# B&R Automation Studio project perfxxl (part 7)

#### referenz.c
```c
#ifdef _DEFAULT_INCLUDES
	#include <AsDefault.h>
#endif
/****************************************************************************/
/*	Ablauf Referenzfahrt */
/*																			*/
/*																			*/
/*	Versionsgeschichte:														*/
/*  Version		Datum		Änderung								von		*/
/*	1.00		25.09.02	erste Implementation					HA		*/
/*	*/
/*		*/
/*																			*/
/****************************************************************************/

#include "glob_var.h"
#include "in_out.h"
#include "standard.h"
#include "motorfunc.h"
#include "auxfunc.h"

#define ROT 0x002D
#define GRUEN 0x000A
#define GRAU 0x0007
#define GRAU59 0x003B
#define SCHWARZ 0x0000
#define WEISS 0x1010

#define RAHMEN_ROT 0x2D00
#define RAHMEN_SCHWARZ 0x0000
#define RAHMEN_GRAU 0x0700

_LOCAL	USINT	ReferenceStep;
_LOCAL TON_10ms_typ ReferenceTimer,CoverLockTimer;
TP_10ms_typ ColorTimer;

_LOCAL	UINT	FeederVerticalColor;
_LOCAL	UINT	FeederHorizontalColor;
_LOCAL	UINT	PaperRemoveVerticalColor;
_LOCAL	UINT	PaperRemoveHorizontalColor;
_LOCAL	UINT	DeloaderHorizontalColor;
_LOCAL	UINT	DeloaderTurnColor;
_LOCAL	UINT	FUColor;
BOOL	ColorToggle;
BOOL	DeloaderReady;
_GLOBAL	UINT	ConveyorBeltOn;
UDINT OriginalDeloaderRefSpeed;
_GLOBAL USINT	ClearLine;
_GLOBAL BOOL	DontCloseTrolley;
/*V1.95 sequenzen disablen, solange Fehlplatte abgeworfen wird*/
_GLOBAL BOOL	DisablePaperRemove;
_GLOBAL UINT MainPicNumber;

static    USINT               PinsStep;       /* holds current step of fct AdjPins */
static    TON_10ms_typ        PinsTimer;

_INIT void Init(void)
{
	PinsStep = 0;
	PinsTimer.IN = FALSE;
	ColorToggle = 0;
	ColorTimer.IN = 1;
	ReferenceStep = 0;
	ReferenceStart = 0;
	ReferenceTimer.IN = 0;
	ReferenceTimer.PT = 1;
	CoverLockTimer.IN = 0;
}

_CYCLIC void Cyclic(void)
{

	SequenceSteps[8] = ReferenceStep;

	TON_10ms(&PinsTimer);

	TON_10ms(&ReferenceTimer);
	TON_10ms(&CoverLockTimer);

	if (!ReferenceStart) ReferenceStep = 0;

	switch (ReferenceStep)
	{
		case 0:
		{

/* wait for start command */
			if (!ReferenceStart) break;

			if(	Motors[FEEDER_VERTICAL].Error
			||	(Motors[FEEDER_HORIZONTAL].Error && GlobalParameter.FlexibleFeeder)
			||	Motors[PAPERREMOVE_VERTICAL].Error
			||	Motors[PAPERREMOVE_VERTICAL2].Error
			||	Motors[PAPERREMOVE_HORIZONTAL].Error
			||	(Motors[DELOADER_HORIZONTAL].Error && GlobalParameter.DeloaderTurnStation>0)
			||	(Motors[DELOADER_TURN].Error && GlobalParameter.DeloaderTurnStation==2) )
			{
				ReferenceStart = 0;
				break;
			}
			ReferenceStep = 100;
			break;
		}

		case 2:
		{

			START = 0;
			PlateTakingStart = 0;
			PaperRemoveStart = 0;
			AdjustStart = 0;
			DeloadStart = 0;
			ExposeStart = 0;
			OpenTrolleyStart = 0;
			CloseTrolleyStart = 0;

			ClearStation(&PlateAtFeeder);
			AdjustReady = 0;
			ExposureReady = 0;
			DeloadReady = 0;
			ClearLine = 0;
			PlateTransportSim = 0;

			Motors[FEEDER_VERTICAL].ReferenceOk = 0;
			Motors[FEEDER_HORIZONTAL].ReferenceOk = 0;
			Motors[PAPERREMOVE_VERTICAL].ReferenceOk = 0;
			Motors[PAPERREMOVE_VERTICAL2].ReferenceOk = 0;
			Motors[PAPERREMOVE_HORIZONTAL].ReferenceOk = 0;
			Motors[DELOADER_HORIZONTAL].ReferenceOk = 0;
			Motors[DELOADER_TURN].ReferenceOk = 0;
			DeloaderReady = 0;
			ReferenceStep = 5;

			break;
		}
		case 5:
		{
			int i;
/*Feeder vacuum off and Feeder vert. reference*/
			for(i=0;i<5;i++)
				Out_FeederVacuumOn[i] = OFF;

			SwitchAdjustTableVacuum(0,ALL,OFF);
			AdjustBlowairOn = 0;
			Out_AdjustSuckerVacuumOn[0] = OFF;
			Out_AdjustSuckerVacuumOn[1] = OFF;
			Out_AdjustSuckerVacuumOn[2] = OFF;
			Out_AdjustSignalCross = OFF;
			Out_LiftingPinsUp = OFF;
			Out_LiftingPinsDown = ON;

			Motors[FEEDER_VERTICAL].StartRef = 1;

/*Deloader Horiz. pre reference very slowly*/
			if(GlobalParameter.DeloaderTurnStation>0)
			{
				Motors[DELOADER_HORIZONTAL].StartRef = 1;
/*HA 02.08.04 V1.80 bugfix: if no turning motor, do not set slow speed*/
				if (GlobalParameter.DeloaderTurnStation==2)
				{
					OriginalDeloaderRefSpeed = Motors[DELOADER_HORIZONTAL].Parameter.ReferenceSpeed;
					Motors[DELOADER_HORIZONTAL].Parameter.ReferenceSpeed = Motors[DELOADER_HORIZONTAL].Parameter.ReferenceSpeed / 2;
				}
			}
			ReferenceStep = 7;
			break;
		}

		case 7:
		{
			if(AdjPins(PINS_DOWN,&PinsStep,&PinsTimer))
				ReferenceStep = 10;
			break;
		}

		case 10:
		{
/*wait for Feeder vert. ref ready, then Feeder Horiz. ref*/

/*if deloader hor is ready, start turn*/
			if(GlobalParameter.DeloaderTurnStation==2)
			{
				if(Motors[DELOADER_HORIZONTAL].ReferenceOk && !Motors[DELOADER_TURN].ReferenceOk)
				{
					Motors[DELOADER_TURN].StartRef = 1;
				}
			}

			if( Motors[FEEDER_VERTICAL].ReferenceOk )
			{
				Out_FeederHorActive = OFF;
				Out_AdjustSuckerActive[0] = OFF;
				Out_AdjustSuckerActive[1] = OFF;
				Out_AdjustSuckerActive[2] = OFF;
				if(GlobalParameter.FlexibleFeeder)
					Motors[FEEDER_HORIZONTAL].StartRef = 1;

				Motors[PAPERREMOVE_VERTICAL].StartRef = 1;
				ReferenceStep = 11;
				break;
			}
			break;
		}

		case 11:
		{
/*X ok? -> start reference*/
			if( !FU.Error && !FU.CANError && FU.ENPO)
			{
				FU.cmd_Ref = 1;
/*wait for reference to start*/
				if(!FU.RefOk)
					ReferenceStep = 12;
			}
			else
				ReferenceStep = 12;
			break;
		}

		case 12:
		{
/*both motors ref ok? -> go on*/
			if(Motors[PAPERREMOVE_VERTICAL].ReferenceOk && Motors[PAPERREMOVE_VERTICAL2].ReferenceOk)
			{
				ReferenceStep = 15;
				break;
			}
/*wait for 1st motor, then start 2nd to avoid current peak*/
			if(Motors[PAPERREMOVE_VERTICAL].ReferenceOk)
			{
				Motors[PAPERREMOVE_VERTICAL2].StartRef = 1;
			}
			break;
		}

		case 15:
		{
/*wait for Feeder Horiz ref  ready, then paper remove vert ref */
/*if deloader hor is ready, start turn*/
			if(GlobalParameter.DeloaderTurnStation==2)
			{
				if(Motors[DELOADER_HORIZONTAL].ReferenceOk && !Motors[DELOADER_TURN].ReferenceOk)
				{
					Motors[DELOADER_TURN].StartRef = 1;
				}
			}
/*if Paperremove vertical ready start horiz*/
			if( Motors[PAPERREMOVE_VERTICAL].ReferenceOk && Motors[PAPERREMOVE_VERTICAL2].ReferenceOk && !Motors[PAPERREMOVE_HORIZONTAL].ReferenceOk )
			{
				Motors[PAPERREMOVE_HORIZONTAL].StartRef = 1;
			}

			if( (Motors[FEEDER_HORIZONTAL].ReferenceOk || !GlobalParameter.FlexibleFeeder) )
			{

				ReferenceStep = 20;
				break;
			}
			break;
		}
		case 20:
		{
/*if deloader hor is ready, start turn*/
			if(GlobalParameter.DeloaderTurnStation==2)
			{
				if(Motors[DELOADER_HORIZONTAL].ReferenceOk && !Motors[DELOADER_TURN].ReferenceOk)
				{
					Motors[DELOADER_TURN].StartRef = 1;
				}
			}

/*wait for Paperrem vert ref ready, then paper remove horiz. ref */
			if( Motors[PAPERREMOVE_VERTICAL].ReferenceOk && Motors[PAPERREMOVE_VERTICAL2].ReferenceOk )
			{
				if( !Motors[PAPERREMOVE_HORIZONTAL].ReferenceOk )
					Motors[PAPERREMOVE_HORIZONTAL].StartRef = 1;
				ReferenceStep = 22;
				break;
			}
			break;
		}
		case 22:
		{

/*if deloader hor is ready, start turn*/
			if(GlobalParameter.DeloaderTurnStation==2)
			{
				if(Motors[DELOADER_HORIZONTAL].ReferenceOk && !Motors[DELOADER_TURN].ReferenceOk)
				{
					Motors[DELOADER_TURN].StartRef = 1;
				}
			}

/*if deloader turn is ready, start hor again*/
			if(GlobalParameter.DeloaderTurnStation==2)
			{
				if(Motors[DELOADER_TURN].ReferenceOk)
				{
					Motors[DELOADER_HORIZONTAL].Parameter.ReferenceSpeed = OriginalDeloaderRefSpeed;
					Motors[DELOADER_HORIZONTAL].ReferenceOk = 0;
					Motors[DELOADER_HORIZONTAL].StartRef = 1;
					ReferenceStep = 23;
				}
			}
			else
				ReferenceStep = 23;

			break;
		}

		case 23:
		{
/*wait for Paperremove horiz. ref ready*/
			if(Motors[PAPERREMOVE_HORIZONTAL].ReferenceOk)
			{
				Out_PaperGripOn[LEFT] = OFF;
				Out_PaperGripOn[RIGHT] = OFF;
				ReferenceStep = 25;
			}
			break;
		}

		case 25:
		{

			switch (GlobalParameter.DeloaderTurnStation)
			{
				case 0:
				{
					ReferenceStep = 45;
					break;
				}
				case 1:
				{
					if (Motors[DELOADER_HORIZONTAL].ReferenceOk)
						ReferenceStep = 45;
					break;
				}
				case 2:
				{
					if (Motors[DELOADER_HORIZONTAL].ReferenceOk && Motors[DELOADER_TURN].ReferenceOk)
						ReferenceStep = 45;
					break;
				}
			}
			break;
		}
		case 45:
		{
/*X ok? -> check if ref ready*/
			if( !FU.Error && !FU.CANError && FU.ENPO)
			{
				if(FU.RefOk)
				{
					ReferenceStep = 46;
				}
			}
/*X not ok? ->ready*/
			else
			{
				ReferenceStep = 50;
			}
			break;
		}

/*HA 10.04.03 new steps 46 and 47 to move to axis parkpos after reference ok*/
/*move X to parkposition*/
		case 46:
		{
			FU.cmd_Park = 1;
			ReferenceStep = 47;
			break;
		}

/*wait for parkposition ready*/
		case 47:
		{
			if(FU.cmd_Park) break;
			ReferenceStep = 50;
			break;
		}

		case 50:
		{
/* Stop Conveyor Belt, Adjuster down */
			if(SendMotorCmd(CONVEYORBELT,"V0",0,0))
			{
				ReferenceStep = 57;
				ConveyorBeltOn = 0;
			}
			break;
		}
		case 57:
		{
			if(!Motors[CONVEYORBELT].Error)
				Motors[CONVEYORBELT].StartRef = 1;

			if( TCPConnected )
				BeamOFF = TRUE;

			ReferenceStep = 60;
			break;
		}
		case 60:
		{
			ClearStation(&PlateAtFeeder);
			AdjustReady = 0;
			ExposureReady = 0;
			DeloadReady = 0;
			PaperRemoveReady = 0;
			ReferenceStep = 0;
			ReferenceStart = 0;
			DontCloseTrolley = 0;
			DisablePaperRemove = 0;
			if(wBildNr == 26)
				wBildNeu = 1;
			break;
		}
/****************************************************************************/
/* HA 26.06.03 V1.11*/
/* SPECIAL STEPS FOR COVER LOCKING/CHECK */
/****************************************************************************/
		case 100:
		{
			if( DoorsOK || UserLevel>=1)
			{
				ReferenceStep = 104;
				CoverLockTimer.IN = 0;
				ReferenceTimer.IN = 0;
				break;
			}
			else
			{
				if(wBildAktuell != 41 )
					OrgBild = wBildAktuell;
				wBildNeu = 41;
				AbfrageOK = 0;
				AbfrageCancel = 0;
				IgnoreButtons = 0;
				OK_CancelButtonInv = 1;
				OK_ButtonInv = 0;
				AbfrageText1 = 43;
				AbfrageText2 = 44;
				AbfrageText3 = 0;
				AbfrageIcon = CAUTION;
				ReferenceStep = 106;
			}
			break;
		}

		case 104:
		{
/*timeout*/
			if( ReferenceTimer.Q )
			{
				CoverLockTimer.IN = 0;
				ReferenceTimer.IN = 0;
				ReferenceStep = 105;
				Out_CoverLockOn = 0;
				break;
			}
/*OK signal in time, or servicelevel 2*/
			if( CoverLockTimer.Q || UserLevel>=1 )
			{
				CoverLockTimer.IN = 0;
				ReferenceTimer.IN = 0;
				ReferenceStep = 2;
				break;
			}
			Out_CoverLockOn = 1;
			CoverLockTimer.IN = CoverLockOK && DoorsOK;
			CoverLockTimer.PT = 100;
			ReferenceTimer.IN = 1;
			ReferenceTimer.PT = 200;
			break;
		}

		case 105:
		{
				if(wBildAktuell != 41 )
					OrgBild = wBildAktuell;
				wBildNeu = 41;
				AbfrageOK = 0;
				AbfrageCancel = 0;
				IgnoreButtons = 0;
				OK_CancelButtonInv = 1;
				OK_ButtonInv = 0;
				AbfrageText1 = 41;
				AbfrageText2 = 42;
				AbfrageText3 = 0;
				AbfrageIcon = CAUTION;
				ReferenceStep = 106;
			break;
		}
/*wait for input */
		case 106:
		{
			if(AbfrageOK)
			{
				AbfrageOK = 0;
				ReferenceStep = 0;
				ReferenceStart = 0;
			}
			break;
		}

	} /*switch*/

/*colors for "LEDs"*/
	ColorTimer.PT = 50;

	if( ColorTimer.IN == 1 && ColorTimer.Q==1)
		ColorTimer.IN = 0;

	if( ColorTimer.IN == 0 && ColorTimer.Q==0)
	{
		ColorToggle = !ColorToggle;
		ColorTimer.IN = 1;
	}

	TP_10ms(&ColorTimer);

	if( Motors[FEEDER_VERTICAL].ReferenceOk)
	{
		FeederVerticalColor = SCHWARZ;
	}
	else
	{
		if(Motors[FEEDER_VERTICAL].Error)
			FeederVerticalColor = GRAU59;
		else
			if(Motors[FEEDER_VERTICAL].StartRef)
			{
				if(ColorToggle)
					FeederVerticalColor = SCHWARZ;
				else
					FeederVerticalColor = WEISS;
			}
			else /*no ref and ref not running*/
				FeederVerticalColor = WEISS;
	}

/*HA 20.01.04 V1.73 */
	if (!GlobalParameter.FlexibleFeeder)
		FeederHorizontalColor = WEISS;
	else
/*END HA 20.01.04 V1.73 */
	if( Motors[FEEDER_HORIZONTAL].ReferenceOk)
	{
		FeederHorizontalColor = SCHWARZ;
	}
	else
	{
		if(Motors[FEEDER_HORIZONTAL].Error)
			FeederHorizontalColor = GRAU59;
		else
			if(Motors[FEEDER_HORIZONTAL].StartRef)
			{
				if(ColorToggle)
					FeederHorizontalColor = SCHWARZ;
				else
					FeederHorizontalColor = WEISS;
			}
			else /*no ref and ref not running*/
				FeederHorizontalColor = WEISS;
	}

	if( Motors[PAPERREMOVE_HORIZONTAL].ReferenceOk)
	{
		PaperRemoveHorizontalColor = SCHWARZ;
	}
	else
	{
		if(Motors[PAPERREMOVE_HORIZONTAL].Error)
			PaperRemoveHorizontalColor = GRAU59;
		else
			if(Motors[PAPERREMOVE_HORIZONTAL].StartRef)
			{
				if(ColorToggle)
					PaperRemoveHorizontalColor = SCHWARZ;
				else
					PaperRemoveHorizontalColor = WEISS;
			}
			else /*no ref and ref not running*/
				PaperRemoveHorizontalColor = WEISS;
	}

	if( Motors[PAPERREMOVE_VERTICAL].ReferenceOk)
	{
		PaperRemoveVerticalColor = SCHWARZ;
	}
	else
	{
		if(Motors[PAPERREMOVE_VERTICAL].Error)
			PaperRemoveVerticalColor = GRAU59;
		else
			if(Motors[PAPERREMOVE_VERTICAL].StartRef)
			{
				if(ColorToggle)
					PaperRemoveVerticalColor = SCHWARZ;
				else
					PaperRemoveVerticalColor = WEISS;
			}
			else /*no ref and ref not running*/
				PaperRemoveVerticalColor = WEISS;
	}

/*HA 20.01.04 V1.73 */
	if (!GlobalParameter.DeloaderTurnStation)
		DeloaderHorizontalColor = WEISS;
	else
/*END HA 20.01.04 V1.73 */
	if( Motors[DELOADER_HORIZONTAL].ReferenceOk)
	{
		DeloaderHorizontalColor = SCHWARZ;
	}
	else
	{
		if(Motors[DELOADER_HORIZONTAL].Error && GlobalParameter.DeloaderTurnStation)
			DeloaderHorizontalColor = GRAU59;
		else
			if(Motors[DELOADER_HORIZONTAL].StartRef)
			{
				if(ColorToggle)
					DeloaderHorizontalColor = SCHWARZ;
				else
					DeloaderHorizontalColor = WEISS;
			}
			else /*no ref and ref not running*/
				DeloaderHorizontalColor = WEISS;
	}

/*HA 20.01.04 V1.73 */
	if (GlobalParameter.DeloaderTurnStation!=2)
		DeloaderTurnColor = WEISS;
	else
/*END HA 20.01.04 V1.73 */
	if( Motors[DELOADER_TURN].ReferenceOk)
	{
		DeloaderTurnColor = SCHWARZ;
	}
	else
	{
		if(Motors[DELOADER_TURN].Error)
			DeloaderTurnColor = GRAU59;
		else
			if(Motors[DELOADER_TURN].StartRef)
			{
				if(ColorToggle)
					DeloaderTurnColor = SCHWARZ;
				else
					DeloaderTurnColor = WEISS;
			}
			else /*no ref and ref not running*/
				DeloaderTurnColor = WEISS;
	}

	if(FU.Error || FU.CANError)
		FUColor = GRAU59;
	else
	if(FU.cmd_Ref && !FU.RefOk)
	{
		if (ColorToggle)
			FUColor = SCHWARZ;
		else
			FUColor = WEISS;
	}
	else
		if(FU.RefOk)
			FUColor = SCHWARZ;
		else
			FUColor = WEISS;

}
```

- motorfunc.h (reference to Logical/GlobalIncludes/motorfunc.h)

#### motorfunc.c
```c
#ifdef _DEFAULT_INCLUDES
	#include <AsDefault.h>
#endif
/*
                             *******************
******************************* C SOURCE FILE *******************************
**                           *******************                           **
**                                                                         **
** project  : LS JET II                                                    **
** filename : MOTORFUNC.C                                                  **
** version  : 1.02                                                         **
** date     : 07.11.2007                                                   **
**                                                                         **
*****************************************************************************
** Abstract                                                                **
** ========                                                                **
** Implementation of motor control functions (sending commands and         **
** check for positions)                                                    **
**                                                                         **
** Copyright (c) 2007, Krause-Biagosch GmbH                                **
** All rights reserved.                                                    **
**                                                                         **
*****************************************************************************
VERSION HISTORY:
----------------
Version     : 1.00
Date        : 20.10.2006
Revised by  : Herbert Aden
Description : Original version.

Version     : 1.01
Date        : 12.10.2007
Revised by  : Herbert Aden
Description : - a variable for holding the current step in function MoveToAbsPosition
                must now be provided by the caller (a pointer to that var of course!)
              - in Fct. IsPositionOK the check for being in a certain position window
                failed, if that window was 0, i.e. if an exact position is to be found
                the expression "currpos - checkpos < deviation" results in false, so it
                was changed to "currpos - checkpos <= deviation" so that if
                currpos==checkpos the result is still true for deviaition==0

Version     : 1.02
Date        : 07.11.2007
Revised by  : Herbert Aden
Description : - bugfix: in RequestMotorData the var SerialCmd.Request was set TRUE
                unconditionally. Caused sporadic Errormessages for serial comm.

*/
#define _MOTORFUNC_C_SRC

/****************************************************************************/
/**                                                                        **/
/**                           INCLUDE FILES                                **/
/**                                                                        **/
/****************************************************************************/
#include <stdlib.h>
#include <string.h>
#include "glob_var.h"
#include "motorfunc.h"

/****************************************************************************/
/**                                                                        **/
/**                       DEFINITIONS AND MACROS                           **/
/**                                                                        **/
/****************************************************************************/
/* NONE */

/****************************************************************************/
/**                                                                        **/
/**                      EXPORTED VARIABLES                                **/
/**                                                                        **/
/****************************************************************************/
/*@checked@*/
_GLOBAL   SerialCmd_Typ       SerialCmd;

/****************************************************************************/
/**                                                                        **/
/**                           GLOBAL VARIABLES                             **/
/**                                                                        **/
/****************************************************************************/
static  BOOL                  Send1Ready = 0;

/****************************************************************************/
/**                                                                        **/
/**                          EXPORTED FUNCTIONS                            **/
/**                                                                        **/
/****************************************************************************/

/****************************************************************************/
/** Send commands to a motor                                                */
/****************************************************************************/
BOOL	SendMotorCmd(const INT pMotor,const char *CmdStr,const BOOL UseValue,const DINT Value)
{
	if(SerialCmd.Send == FALSE) /*wait, till no other sending active*/
	{
		strcpy(SerialCmd.CmdString,CmdStr);
		SerialCmd.UseParameter = UseValue;
		SerialCmd.Parameter = Value;
		if (   (STREQ(CmdStr,CMD_ABSOLUTE_POS))
			|| (STREQ(CmdStr,CMD_RELATIVE_POS))
			|| (STREQ(CmdStr,CMD_MOVE_AT))
		  ) /*bei LA oder LR oder V Refdir verwenden, sonst nicht*/
			SerialCmd.UseRefDirection = TRUE;
		else
			SerialCmd.UseRefDirection = FALSE;

		SerialCmd.SendMotor = pMotor;
		SerialCmd.Send = TRUE;
		return TRUE;
	}
	else
		return FALSE;
}

/****************************************************************************/
/** Request data from a motor                                                */
/****************************************************************************/
BOOL	RequestMotorData(const INT pMotor,const char *CmdString)
{
	if( SerialCmd.Send == TRUE )
		return FALSE;
	else
	{
		SerialCmd.Request = TRUE;
		return SendMotorCmd(pMotor,CmdString,FALSE,0);
	}
}

/****************************************************************************/
/** Check, if a motor is in a certain position window                       */
/****************************************************************************/
BOOL	isPositionOk(const INT Motor,const DINT Pos,const DINT Deviation)
{
	DINT tmp;
	if (labs(Deviation) > 0 )
		tmp = labs(Deviation);
	else	/* if Dev is 0, then use deviation defined in motorparam*/
		tmp = labs(Motors[Motor].Parameter.PositionWindow);

	if( labs( labs(Motors[Motor].Position) - labs(Pos) ) <= tmp )
		return TRUE;
	else
		return FALSE;
}

/****************************************************************************/
/** Check, if a motor is below a certain position                           */
/****************************************************************************/
BOOL	isPositionLowerThan(const INT Motor,DINT Pos)
{
	if( labs(Motors[Motor].Position) < (labs(Pos) ) )
		return TRUE;
	else
		return FALSE;
}

/****************************************************************************/
/** Check, if a motor is above a certain position                           */
/****************************************************************************/
BOOL	isPositionHigherThan(const INT Motor,DINT Pos)
{
	if( labs(Motors[Motor].Position) > (labs(Pos) ) )
		return TRUE;
	else
		return FALSE;
}

/****************************************************************************/
/* send commands to paper remove vertical */
/****************************************************************************/
BOOL	PapRemVerticalCmd(BOOL Config,char *CmdString,BOOL UseValue,DINT Value)
{
	if(Config == LEFT)
		return SendMotorCmd(PAPERREMOVE_VERTICAL, CmdString, UseValue, Value);
	else
	if(Config == RIGHT)
		return SendMotorCmd(PAPERREMOVE_VERTICAL2, CmdString, UseValue, Value);
	else
	if ( Send1Ready == FALSE )
	{
		if( SendMotorCmd(PAPERREMOVE_VERTICAL, CmdString, UseValue, Value) )
			Send1Ready = TRUE;

		return FALSE;
	}
	else
	{
		if( SendMotorCmd(PAPERREMOVE_VERTICAL2, CmdString, UseValue, Value) )
		{
			Send1Ready = FALSE;
			return TRUE;
		}
		return FALSE;
	}
}

/****************************************************************************/
/* Check position of paper remove vertical */
/****************************************************************************/
BOOL	isPapRemVerticalOk(BOOL Config,DINT Pos,UDINT MaxDeviation)
{
	if(Config == LEFT)
		return isPositionOk(PAPERREMOVE_VERTICAL, Pos, MaxDeviation);
	else
	if(Config == RIGHT)
		return isPositionOk(PAPERREMOVE_VERTICAL2, Pos, MaxDeviation);
	else
	if ( isPositionOk(PAPERREMOVE_VERTICAL, Pos, MaxDeviation) )
	{
		if ( isPositionOk(PAPERREMOVE_VERTICAL2, Pos, MaxDeviation) )
			return TRUE;
		else
			return FALSE;
	}
	else
		return FALSE;
}

/****************************************************************************/
/* move motor to an absolute position and wait for motion to start */
/****************************************************************************/
BOOL  MoveToAbsPosition(INT pMotor, DINT Pos, DINT Speed, USINT *pStep)
{
	int step = *pStep;

	BOOL retval = FALSE;

	if (pMotor == 0 && Pos == 0L && Speed == 0L)
	{
		step = 0;
		*pStep = 0;
		return FALSE;
	}

	switch (step)
	{
		case 0:
		{
/* send target position */
			if( SendMotorCmd(pMotor,CMD_ABSOLUTE_POS,TRUE,Pos) )
			{
				if ( Speed == DONT_SEND_SPEED )
					step = 20;
				else
					step = 10;
			}
			retval = FALSE;
			break;
		}
/* set speed */
		case 10:
		{
			if( SendMotorCmd(pMotor,CMD_SPEED,TRUE,Speed) )
			{
				step = 20;
			}
			retval = FALSE;
			break;
		}
		case 20:
		{
/* start motion */
			if( SendMotorCmd(pMotor,CMD_START_MOTION,FALSE,0L) )
			{
				step = 30;
			}
			retval = FALSE;
			break;
		}
		case 30:
		{
/* Wait til motion begins or Motor is in position (might be already there!)*/
			if( Motors[pMotor].Moving
			    ||
			    isPositionOk(pMotor,Pos,0) )
			{
				step = 0;
				retval = TRUE;
			}
			break;
		}
	}
	*pStep = step;
	return retval;
}

/****************************************************************************/
/* move motor to an relative position without waiting for motion to start */
/****************************************************************************/
BOOL  MoveToRelPosition(INT pMotor, DINT Pos, DINT Speed, USINT *pStep)
{
	int step = *pStep;

	BOOL retval = FALSE;

	if (pMotor == 0 && Pos == 0L && Speed == 0L)
	{
		step = 0;
		*pStep = 0;
		return FALSE;
	}

	switch (step)
	{
		case 0:
		{
/* send target position */
			if( SendMotorCmd(pMotor,CMD_RELATIVE_POS,TRUE,Pos) )
			{
				if ( Speed == DONT_SEND_SPEED )
					step = 20;
				else
					step = 10;
			}
			retval = FALSE;
			break;
		}
/* set speed */
		case 10:
		{
			if( SendMotorCmd(pMotor,CMD_SPEED,TRUE,Speed) )
			{
				step = 20;
			}
			retval = FALSE;
			break;
		}
		case 20:
		{
/* start motion */
			if( SendMotorCmd(pMotor,CMD_START_MOTION,FALSE,0L) )
			{
				step = 30;
			}
			retval = FALSE;
			break;
		}
		case 30:
		{
			step = 0;
			retval = TRUE;
			break;
		}
	}
	*pStep = step;
	return retval;
}

/****************************************************************************/
/**                                                                        **/
/**                          LOCAL FUNCTIONS                               **/
/**                                                                        **/
/****************************************************************************/
/* NONE */

/****************************************************************************/
/**                                                                        **/
/**                                 EOF                                    **/
/**                                                                        **/
/****************************************************************************/
```

- auxfunc.h (reference to Logical/GlobalIncludes/auxfunc.h)

### Program Logical/Exposer/Ablauf/expose (ANSIC, version 1.12.0) - Belichtungsablauf

#### belichten.c
```c
#ifdef _DEFAULT_INCLUDES
	#include <AsDefault.h>
#endif
/****************************************************************************/
/*	Ablauf belichten */
/*																			*/
/*																			*/
/*	Versionsgeschichte:														*/
/*  Version		Datum		Änderung								von		*/
/*	1.0			19.09.02	erste Implementation					HA		*/
/*	1.10		13.11.02	erweiterte TB1-Komm. (Polygonspeed)		HA		*/
/*	1.11		02.04.03	Belichtung wird im AUTO Modus nicht 	HA		*/
/*							gestartet, wenn keine Verbindung zum TIFFBlaster */
/*							und keine TB Simulation*/
/*	1.12		07.04.03	Ausgabe: Warte auf Daten..." implementiert 	HA		*/
/*																			*/
/*																			*/
/****************************************************************************/

#include "glob_var.h"
#include "asstring.h"
#include "sys_lib.h"
#include "in_out.h"
#include <string.h>

#define	MAXFILELIST	32
#define TCPIPTIMEOUT 150

_LOCAL	USINT	ExposeStep;
_LOCAL TON_10ms_typ ExposeTimer;
USINT			tmp[20];

_GLOBAL	STRING	FileName[100];
_GLOBAL	USINT	FileListShift;
_GLOBAL	STRING	FileListName[MAXFILELIST][50];
_GLOBAL	STRING	FileListStatus[MAXFILELIST][5];
_GLOBAL	STRING	FileListTime[MAXFILELIST][20];
_GLOBAL	STRING	FileListResolution[MAXFILELIST][5];

_GLOBAL BOOL	AdjustFailed;
_GLOBAL BOOL	ExposingStarted;	/*HA 08.07.03 V1.14 Flag to inform plate taking that exposing has started*/

_GLOBAL	RTCtime_typ	RTCtime;

_GLOBAL UDINT	PlatesMade;		/* [0] = Plates made ever,[1] = plates made today*/
_GLOBAL	UDINT	PlatesMadeToday;
_GLOBAL	BOOL	savePlatesMade;

_GLOBAL USINT	ClearLine;

_LOCAL	USINT	Length,PermanentMode;

int	TimeoutCounter,i;
BOOL	StepChanged;
_LOCAL UINT	ExposureProgress;
_GLOBAL 	BOOL	SendYOffset,SendLP,SendOSCommand;
STRING tmpstr[100];
int waitcounter;

_LOCAL    UINT                CheckForDataStep;
_LOCAL    USINT               TestNumberOfPlates,TestPlateType;
static    USINT               OldSecond;
_LOCAL    BOOL                StopCheckingForData;

_INIT void init(void)
{
	StepChanged = 0;
	ExposeStep		= 0;
	ExposeStart	= 0;
	ExposureReady		= 0;
	ExposeTimer.IN	= 0;
	ExposeTimer.PT	= 10; /*just to have any value in there...*/

	Expose_Param.ScansPerMinute			= 96000;
	Expose_Param.Resolution				= 1270;

	PlatesMadeToday = 0;
	ExposingStarted = 0;
	PermanentMode = 0;
	CheckForDataStep = 0;
	StopCheckingForData = 0;
	OldSecond = 0;
	TestPlateType = 1;
}

_CYCLIC void cyclic(void)
{
UINT RequiredLaserPower;

	SequenceSteps[4] = ExposeStep;

	TON_10ms(&ExposeTimer);

/*	if(START)*/
/*HA 28.05.03 V1.13 added "|| ClearLine" */
	if( (AdjustReady) && AUTO
		&& (GlobalParameter.TBSimulation || TCPConnected || ClearLine))
		 ExposeStart=1;

/*safety*/
	if( !ExposeStart )
	{
		 PermanentMode = 0;
		 ExposeStep = 0;
		 ExposingStarted = 0;
/*		 strcpy(FileName,"----");*/
		 ExposureProgress = 0;
	}

	switch (ExposeStep)
	{
		case 0:
		{
			if(!ExposeStart) break;

			ExposeStep = 2;
			break;
		}

		case 2:
		{
			REAL AccWay = 3.0;
			if (DisableTable || AdjustStart) break; /*SAFETY*/

/* for LSJet 350: if speed is > than the usual 97000 then double acceleration/deceleration way*/
			if(Expose_Param.ScansPerMinute < 99000)
				AccWay = 3.0;
			else
				AccWay = 6.0;

			Expose_Param.PEGStartPosition = PlateParameter.XOffset+PlateParameter.Length;
			if ( Expose_Param.PEGStartPosition > X_Param.MaxPosition ) Expose_Param.PEGStartPosition = X_Param.MaxPosition;
			Expose_Param.PEGEndPosition = PlateParameter.XOffset;
			if ( Expose_Param.PEGEndPosition < X_Param.MinPosition ) Expose_Param.PEGEndPosition = X_Param.MinPosition;
			Expose_Param.StartPosition = PlateParameter.XOffset+PlateParameter.Length + AccWay;
			if ( Expose_Param.StartPosition > X_Param.MaxPosition ) Expose_Param.StartPosition = X_Param.MaxPosition;
			Expose_Param.EndPosition = PlateParameter.XOffset - AccWay;
			if ( Expose_Param.EndPosition < X_Param.MinPosition ) Expose_Param.EndPosition = X_Param.MinPosition;

			if ( FU.cmd_Target == 0 )
			{
				FU.TargetPosition_mm = Expose_Param.StartPosition;
				FU.cmd_Target = 1;
				ExposeStep = 3;
			}
			break;
		}
		case 3:
		{
/*und warten*/
			if ( abs(FU.aktuellePosition_mm - FU.TargetPosition_mm )< 2 )
			{
/*Tisch ist in Position -> OK, weiter*/
				ExposeStep = 5;
			}
			break;
		}

		case 5:
		{
/* Communication with TiffBlaster*/
			if(GlobalParameter.TBSimulation || ClearLine)
			{
				strcpy(FileName,"KrauseTestImage.TIF");
				ExposeStep = 20;
				StepChanged = 1;
				break;
			}
/*Warte auf Daten...*/
			if (DataReady)
			{
				ExposeStep = 15;
				StepChanged = 1;
				StopCheckingForData = 1;
			}

			break;
		}

/*V2.15 automatische Laserleistungseinstellung bei Aufl Wechsel*/
		case 15:
		{
			if( AdjustFailed  )
			{
				ExposeStep	= 0;
				ExposeStart	= 0;
				break;
			}

/*
if plate is longer than 600 mm then wait for adjusting to finish,
to make sure, the plate cannot be under the beam during power setting
*/
			if(!AdjustReady && AUTO && (PlateParameter.Length>600))
				break;

/*Range check for safety*/
			if(Expose_Param.Resolution < 300 || Expose_Param.Resolution > 4000)
			{
				Expose_Param.Resolution=1270;
				GlobalParameter.Resolution = 1270;
			}

/*check, which laserpower to use*/
			RequiredLaserPower = GlobalParameter.RealLaserPower;
/*gehe durch die Liste, bis sie entweder ganz abgearbeitet ist oder die passende Aufl gefunden wurde*/
			for (i=1; i<MAXLASERPOWERSETTINGS ; i++)
			{
				if ( Expose_Param.Resolution == LaserPowerSettings[i].Resolution )
				{
/*if-construct for safety*/
					if ((PlateParameter.Number>0)&& (PlateParameter.Number<MAXPLATETYPES))
						RequiredLaserPower = LaserPowerSettings[i].LaserPower[PlateParameter.Number];
					else
						RequiredLaserPower = LaserPowerSettings[i].LaserPower[1];
					break;
				}
			}

/*if the power is different from currently used power, then send new power*/
			if (RequiredLaserPower != GlobalParameter.RealLaserPower)
			{
				GlobalParameter.RealLaserPower = RequiredLaserPower;
				SendLP = 1;
			}

/*go ahead if Power setting is ready or not started*/
			if ( !SendLP )
			{
				ExposeStep = 16;
/* HA V1.36 08.05.06 send Open Shutter command to TB*/
				SendOSCommand = 1;
				StepChanged = 1;
			}
			break;
		}

/* HA V2.10  08.05.06 send Open Shutter command to TB*/
		case 16:
		{
			waitcounter = 0;
			if (SendOSCommand == 0)
				ExposeStep = 18;
			break;
		}

/* wait shortly*/
		case 18:
		{
			waitcounter++;
			if (waitcounter >= 120)/*120 cycles = 0,6 sec*/
			{
				ExposeStep = 20;
				waitcounter = 0;
				StepChanged = 1;
			}
			break;
		}

		case 20:
		{
			if(StepChanged)
			{
				if(strlen(FileName)<50)
					strcpy(&FileListName[MAXFILELIST-1][0],FileName);
				else
				{
					memcpy(&FileListName[MAXFILELIST-1][0],FileName,48);
					FileListName[MAXFILELIST-1][49]=0;
				}
				itoa(Expose_Param.Resolution,(UDINT)&FileListResolution[MAXFILELIST-1][0]);
				strcpy(&FileListStatus[MAXFILELIST-1][0],"ACT");
				itoa(RTCtime.hour,(UDINT)&tmp[0]);
				if(RTCtime.hour<=9)
					strcpy(&FileListTime[MAXFILELIST-1][0],"0");
				else
					strcpy(&FileListTime[MAXFILELIST-1][0],"");
				strcat(&FileListTime[MAXFILELIST-1][0],&tmp[0]);
				strcat(&FileListTime[MAXFILELIST-1][0],":");
				itoa(RTCtime.minute,(UDINT)&tmp[0]);
				if(RTCtime.minute<=9)
					strcat(&FileListTime[MAXFILELIST-1][0],"0");
				strcat(&FileListTime[MAXFILELIST-1][0],&tmp[0]);
				strcat(&FileListTime[MAXFILELIST-1][0],":");
				itoa(RTCtime.second,(UDINT)&tmp[0]);
				if(RTCtime.second<=9)
					strcat(&FileListTime[MAXFILELIST-1][0],"0");
				strcat(&FileListTime[MAXFILELIST-1][0],&tmp[0]);
				StepChanged = 0;
				FileListShift = 1;
			}

			if(Expose_Param.Resolution < 300 || Expose_Param.Resolution > 4000)
			{
				Expose_Param.Resolution=1270;
				GlobalParameter.Resolution = 1270;
			}

			if(Expose_Param.ScansPerMinute<1000 || Expose_Param.ScansPerMinute>150000)
				Expose_Param.ScansPerMinute = 76200;

/*calculate X-speed*/
			Expose_Param.ExposeSpeed = (25.4/60.0) * ((REAL)Expose_Param.ScansPerMinute/(REAL)Expose_Param.Resolution);

			if(Expose_Param.ExposeSpeed<1 || Expose_Param.ExposeSpeed>100)
				Expose_Param.ExposeSpeed = 25.4;

/*wait for adjusting to finish*/
			if( AdjustReady || !AUTO)
			{
				FU.cmd_Expose = 1;
/*HA 08.07.03 V1.14 Flag to inform plate taking that exposing has started*/
				ExposingStarted = 1;
				ExposeStep = 25;
				StepChanged = 1;
			}

/*HA 17.02.04 V1.74B Adjusting failed and MaxFailedPlates is 0: stop */
			if( AdjustFailed && (AdjusterParameter.MaxFailedPlates == 0) )
			{
				ExposeStep	= 0;
				ExposeStart	= 0;
				break;
			}

			if( AdjustFailed && AUTO )
			{
				strcpy(&FileListStatus[0][0],"ERR");
				itoa(RTCtime.hour,(UDINT)&tmp[0]);
				if(RTCtime.hour<=9)
					strcpy(&FileListTime[0][0],"0");
				else
					strcpy(&FileListTime[0][0],"");
				strcat(&FileListTime[0][0],&tmp[0]);
				strcat(&FileListTime[0][0],":");
				itoa(RTCtime.minute,(UDINT)&tmp[0]);
				if(RTCtime.minute<=9)
					strcat(&FileListTime[0][0],"0");
				strcat(&FileListTime[0][0],&tmp[0]);
				strcat(&FileListTime[0][0],":");
				itoa(RTCtime.second,(UDINT)&tmp[0]);
				if(RTCtime.second<=9)
					strcat(&FileListTime[0][0],"0");
				strcat(&FileListTime[0][0],&tmp[0]);

				ExposureReady = 1;
				ExposeStep = 26;
			}
			break;
		}

		case 25:
		{
#ifdef PERFORMANCE
			if ((FU.aktuellePosition_mm <= Expose_Param.PEGStartPosition) && (PlateParameter.Length > 1))
			{
				ExposureProgress = ((Expose_Param.PEGStartPosition - FU.aktuellePosition_mm) *100.0)
									 / PlateParameter.Length;
			}
#else
			if ((FU.aktuellePosition_mm > Expose_Param.PEGStartPosition) && (PlateParameter.Length > 1))
			{
				ExposureProgress = ((FU.aktuellePosition_mm-Expose_Param.PEGStartPosition) *100.0)
									 / PlateParameter.Length;
			}
#endif
			else
				ExposureProgress = 0;
/*Wait for Exposure ready*/
			if(FU.cmd_Expose) break;
			if(!ExposureReady)
			{
				strcpy(&FileListStatus[0][0],"RDY");
				itoa(RTCtime.hour,(UDINT)&tmp[0]);
				if(RTCtime.hour<=9)
					strcpy(&FileListTime[0][0],"0");
				else
					strcpy(&FileListTime[0][0],"");
				strcat(&FileListTime[0][0],&tmp[0]);
				strcat(&FileListTime[0][0],":");
				itoa(RTCtime.minute,(UDINT)&tmp[0]);
				if(RTCtime.minute<=9)
					strcat(&FileListTime[0][0],"0");
				strcat(&FileListTime[0][0],&tmp[0]);
				strcat(&FileListTime[0][0],":");
				itoa(RTCtime.second,(UDINT)&tmp[0]);
				if(RTCtime.second<=9)
					strcat(&FileListTime[0][0],"0");
				strcat(&FileListTime[0][0],&tmp[0]);
				StepChanged = 0;
				PlatesMade++;
				PlatesMadeToday++;
				savePlatesMade=1;
			}
			ExposureReady = 1;
			ExposeStep = 26;
			ExposureProgress = 0;

			StopCheckingForData = 0;
			DataReady = 0;
			break;
		}
		case 26:
		{

/*feeder fährt runter: Tisch darf nicht fahren*/
			if (DisableTable)
				break;

/****************************************************************************/

/*wait for deloading ready, then go on*/
			if(DeloadReady || !AUTO)
			{
				DeloadReady = 0;
				ExposureReady = 0;
				ExposeStep = 30;
			}

			break;
		}
		case 30:
		{
			if ( PermanentMode && !AUTO )
				ExposeStep = 5;
			else
				ExposeStep = 35;
			break;
		}
		case 35:
		{
			ExposeStep = 0;
			ExposeStart = 0;
			break;
		}
	} /*switch*/

/****************************************************************************/
/* V2.50 asynchronous checking for data*/
/****************************************************************************/
	if( (ReferenceStart && (ExposeStep == 0))
	 || (ClearLine == TRUE)
	)
	{
		DataReady = 0;
		StopCheckingForData = 0;
		CheckForDataStep = 0;
	}

	if(GlobalParameter.TBSimulation)
	{
/* V2.55 Durchlaufsimulation*/
		DataReady = 1;
		TestNumberOfPlates = 3;

		if (TestNumberOfPlates==0)
			TestNumberOfPlates = 1;
		if (DataReady)
		{
			PlateToDo.PlateType = TestPlateType;
		}

	}

	switch (CheckForDataStep)
	{
		case 0:
		{
/*	check for data every second */
			if( (RTCtime.second != OldSecond)
			&& !StopCheckingForData
			&& !(GlobalParameter.TBSimulation || !TCPConnected)
			&& !ClearLine
			&& !SendLP
			&& !SendOSCommand
			&& !SendYOffset
			&& !ReferenceStart
			  )
				CheckForDataStep = 5;
			break;
		}
		case 5:
		{
/* Communication with TiffBlaster*/
			OldSecond = RTCtime.second;
			if(TCPSendCmd == 0)
			{
				strcpy(TCPCmd,"15");
				TCPSendCmd = 1;
				CheckForDataStep = 6;
			}
			TimeoutCounter = 0;
			break;
		}
		case 6:
		{

			if( !TCPRcvFlag)
			{
				TimeoutCounter++;
				if(TimeoutCounter>TCPIPTIMEOUT)
				{
					TimeoutCounter = 0;
					if(GlobalParameter.TBSimulation || !TCPConnected)
					{
						CheckForDataStep = 0;
						break;
					}

					CheckForDataStep = 0;
					DataReady = 0;
					switch (GlobalParameter.Language)
					{
						case 0:
						{
							strcpy(FileName,"Warte auf TIFF Blaster...");
							break;
						}
						case 1:
						{
							strcpy(FileName,"Waiting for TIFF Blaster...");
							break;
						}
					}
				}
				break;
			}

/*****       TCP answer received   *************/
/*IP0 : wait*/
			TCPRcvFlag = 0;
			if( TCPAnswer[2]=='0')
			{
				CheckForDataStep = 7;
				TimeoutCounter = 0;
				DataReady = 0;
				switch (GlobalParameter.Language)
				{
					case 1: /*deutsch*/
					{
						strcpy(FileName,"Warte auf Daten...");
						break;
					}
					default: /*english*/
					{
						strcpy(FileName,"Waiting for data...");
					}
				}
				break;
			}
			if(TCPAnswer[2]=='1')
			{
/* Aufbau des Strings:

Byte 0..2 	Fix: IP1
Byte 3..6 	Auflösung, fix 4stellig
Byte 7..12	Scans Pro Minute, fix 6stellig
Byte 13		Plattentyp
Byte 14		Anzahl Platten
Byte 15..End	Dateiname
BSP:	IP1127009600032C:\FileName.TIF
*/

				Length = strlen(TCPAnswer)-15;
				if(Length < 50 && Length>0 )
				{
			/*extract resolution*/
					memcpy(	tmp,&TCPAnswer[3],4 );
					tmp[4] = 0;
					Expose_Param.Resolution = atoi((UDINT) &tmp);
			/*extract Scans per min */
					memcpy(	tmp,&TCPAnswer[7],6 );
					tmp[6] = 0;
					Expose_Param.ScansPerMinute = atoi((UDINT) &tmp);
			/*extract Platetype */
					memcpy(	tmp,&TCPAnswer[13],1 );
					tmp[1] = 0;
			/*extract Number of plates */
					memcpy(	tmp,&TCPAnswer[14],1 );
					tmp[1] = 0;
			/*extract Filename */
					memcpy(	FileName,&TCPAnswer[15],Length );
					FileName[Length]=0;
				}
				CheckForDataStep = 0;
				DataReady = 1;
				StopCheckingForData = 1;
			}
			break;
		}

/*Warteschritt, um 14 etwas langsamer zu schicken*/
		case 7:
		{
/*Timeoutcounter hier als wartecounter missbraucht*/
			TimeoutCounter++;
			if(TimeoutCounter>20) /* 200 ms*/
			{
				TimeoutCounter = 0;
				CheckForDataStep = 5;
			}
			break;
		}
	}

}
```

### Program Logical/Exposer/Ablauf/entladen (ANSIC, version 1.30.0) - Platte Entladen aufs Transportband

#### entladen.c
```c
#ifdef _DEFAULT_INCLUDES
	#include <AsDefault.h>
#endif
/****************************************************************************/
/*	Ablauf Platte Entladen */
/*																						*/
/*																						*/
/*	Versionsgeschichte:																*/
/*  Version		Datum		Änderung										von		*/
/*	1.0			17.09.02	erste Implementation								HA		*/
/*																						*/
/*																						*/
/****************************************************************************/
#include "glob_var.h"
#include "asstring.h"
#include <string.h>
#include "in_out.h"
#include "Motorfunc.h"
#include "auxfunc.h"

#define CONVEYORBELT_BACKWAY	5000

_LOCAL	USINT	DeloadStep;
_LOCAL TON_10ms_typ DeloadTimer;
USINT			tmp[20];

_LOCAL TON_10ms_typ CycleTimer,CycleTimer2,TestTimer;
_LOCAL R_TRIGtyp R_TRIG_01;
_LOCAL F_TRIGtyp F_TRIG_01,F_TRIG_02;

BOOL	Started;
_GLOBAL UDINT PlatesPerHour;
/*HA 21.01.04 V1.73*/
_GLOBAL BOOL	AdjustFailed;

_LOCAL	UINT	CurrentTime;
_LOCAL	REAL	LastTime,HandlingTime;
DINT	Result1,Result2;
UDINT	TurnSpeedOld;
		TOF_10ms_typ	ConveyorBeltDelay;
		TON_10ms_typ	EGMErrorDelay;
		TON_10ms_typ	PinsDownWait;
		TON_10ms_typ	TurnOK;
		TOF_10ms_typ	ConveyorBeltSensorDelay1,ConveyorBeltSensorDelay2;

_GLOBAL	UINT			ConveyorBeltOn;

/*HA 14.01.04 V1.71 implemented Stop pins on conveyor */
_GLOBAL	BOOL			StopPinsUp;
		TON_10ms_typ	PinsDownDelay;
		TOF_10ms_typ	PinsUpDelay;

/*HA 05.09.03 V1.51 to avoid adjustsensor triggered by deloaded plate*/
/*HA 08.09.03 V1.52 disable-flags for right adjuster*/
_GLOBAL 	BOOL			DisableAdjustSensor,DisableAdjusterUp,EnableShuttle;
_LOCAL	BOOL			StartConveyorBelt,StopConveyorBelt;
		BOOL			LayOffPos2;
		UDINT			TempPlateReleasePosition,TempTurnPosition,TempTakePosition;

		REAL			PlateDeloadLength; /*holds calculated value Length*LengthFactor*/
BOOL TurnPosOK; /*Hilfsvariable für drehen ohne Zeit*/
_GLOBAL	BOOL	ConveyorbeltSimulation;
int DeloadSpeed,StopPinsStep;
BOOL	DisableConveyorBelt;
DINT ConveyorBeltPos,ConveyorBeltBack;
BOOL dummyflag;
USINT	ReturnStep;
_GLOBAL UINT	HideKrause;
USINT ConveyorBeltStep;
TON_10ms_typ	ConveyorBeltTimer;
UDINT	ConveyorTime;

_GLOBAL	REAL	TablePosDrop;
BOOL	MovingToParkpos,NoSpeedChange;
static USINT ConvMotStep;
TON_10ms_typ LiftpinsDownTimer;
static BOOL FirstTime;
static REAL OldParkSpeed;
static BOOL ParkSpeedChanged;

_LOCAL BOOL  JetValuesValid;
_LOCAL REAL  JetSqmValue; /* in m² for the plate set, i.e. no matter if 1 or 2 plates,
                             sum up must be done by jet */
_LOCAL USINT JetPlateCnt; /* 1 or 2 plates*/
static TON_10ms_typ JetValuesValidDelay;

void InformBluefin(void)
{
	if(!JetValuesValid)
	{
		if(PlateOnConveyorBelt.PlateConfig == BOTH)
			JetPlateCnt = 2;
		else
			JetPlateCnt = 1;

		if( (PlateOnConveyorBelt.PlateType > 0)
		 && (PlateOnConveyorBelt.PlateType < MAXPLATETYPES)
		  )
		{
/* /1000 weil Length und Width in mm sind, die Fläche aber in QadratMETER*/
			JetSqmValue = (PlateTypes[PlateOnConveyorBelt.PlateType].Length / 1000.0) *
			              (PlateTypes[PlateOnConveyorBelt.PlateType].Width / 1000.0);
				JetSqmValue *= JetPlateCnt;
		}
/* little delay to make sure the values are transmitted before the valid flag is set*/
		JetValuesValidDelay.IN = TRUE;
	}
	/* no else: Bluefin did not reset Valid-flag...do nothing */
}

_INIT void init(void)
{
	JetValuesValidDelay.IN = FALSE;
	JetValuesValid = FALSE;
	JetSqmValue = 0.0;
	JetPlateCnt = 1;
	ParkSpeedChanged = FALSE;
	FirstTime = TRUE;
	ConvMotStep = 0;
	LayOffPos2 = 0;
	ClearStation(&PlateOnConveyorBelt);
	DisableConveyorBelt = 0;
	StopPinsStep = 0;
	ClearStation(&PlateAtDeloader);
	TurnSpeedOld	= 0;
	DeloadStep		= 0;
	DeloadStart	= 0;
	DeloadReady		= 0;
	DeloadTimer.IN	= 0;
	DeloadTimer.PT	= 10; /*just to have any value in there...*/
	CycleTimer.IN	= 0;
	CycleTimer.PT	= 10; /*just to have any value in there...*/
	ConveyorBeltDelay.IN = 0;
	ConveyorBeltDelay.PT = 1000;
	ConveyorBeltOn = FALSE;
	EnableShuttle = 0;
	TurnOK.PT = 50;
	TurnOK.IN = 0;
	TurnPosOK = 0;
	LiftpinsDownTimer.IN = FALSE;

}

/****************************************************************************/
/* zyklischer Teil*/
/****************************************************************************/
_CYCLIC void cyclic(void)
{
#ifdef PERFORMANCE
	GlobalParameter.DeloaderTurnStation = 0;
#endif

	if( GlobalParameter.DisableSlowMode )
		SlowMode = 0;
	if( GlobalParameter.SlowModeWaitTime > 9900 )
		GlobalParameter.SlowModeWaitTime = 2000;

	SequenceSteps[5] = DeloadStep;

	if(ExposureReady && AUTO)
		DeloadStart = 1;

	TON_10ms(&DeloadTimer);
	TON_10ms(&TurnOK);

	LiftpinsDownTimer.IN = Out_LiftingPinsDown;
	LiftpinsDownTimer.PT = 12000; /* 2 min */
	TON_10ms(&LiftpinsDownTimer);

/* little delay for Bluefin comm handshake flag*/
	JetValuesValidDelay.PT = 15; /* 150ms */
	TON_10ms(&JetValuesValidDelay);
	if(JetValuesValidDelay.Q)
	{
		JetValuesValidDelay.IN = FALSE;
		JetValuesValid = TRUE;
	}
/* time measurement*/

/*detect edge of expose command*/
R_TRIG_01.CLK = FU.cmd_Expose;
R_TRIG(&R_TRIG_01);
if(R_TRIG_01.Q && Started)
{
	Started = 0;
	CycleTimer.IN = 0;
	Result1 = CycleTimer.ET;
	CycleTimer2.IN = 1;
	LastTime = (REAL)(Result1)/100.0;
	PlatesPerHour = (UDINT) ((3600.0 / ( ((REAL) (Result1))/100.0))+0.5);
}
else
if(R_TRIG_01.Q && !Started)
{
	Started = 1;
	CycleTimer.IN = 1;
	CycleTimer2.IN = 0;
	Result2 = CycleTimer2.ET;
	LastTime = (REAL)(Result2)/100.0;
	PlatesPerHour = (UDINT) ((3600.0 / ( ((REAL) (Result2))/100.0))+0.5);
}

if(CycleTimer.IN)
{
	CurrentTime = CycleTimer.ET;
}
if(CycleTimer2.IN)
{
	CurrentTime = CycleTimer2.ET;
}

CycleTimer.PT = 60000; /*max 1 min*/
TON_10ms(&CycleTimer);
CycleTimer2.PT = 60000; /*max 1 min*/
TON_10ms(&CycleTimer2);

/*time measurement handling time (end of exposure to start of exposure*/
TestTimer.IN = !FU.cmd_Expose;
if( TestTimer.IN )
{
	HandlingTime = ((REAL) TestTimer.ET) / 100.0;
}
TestTimer.PT = 60000;
TON_10ms(&TestTimer);

/*safety*/
	if( !DeloadStart )
	{
		DeloadStep = 0;
		DisableAdjustSensor = 0;
		EnableShuttle = 0;
		MovingToParkpos = FALSE;
		if(ParkSpeedChanged)
		{
			X_Param.ParkSpeed = OldParkSpeed;
			ParkSpeedChanged = FALSE;
		}

	}

	switch (DeloadStep)
	{
		case 0:
		{
			if( !DeloadStart
			 ||  AdjustStart
			  )
				break;

			DeloadTimer.IN = 0;
			DeloadStep = 1;
/*HA 05.09.03 V1.51 to avoid adjustsensor triggered by deloaded plate*/
			DisableAdjustSensor = 0;

			break;
		}
		case 1:
		{
/*Wait for Exposure to finish*/
			if(ExposureReady || !ExposeStart || !AUTO)
			{
				DeloadStep = 170;
				break;
			}

			break;
		}

/****************************************************************************/
/*Deloading without turn/positioning device*/
/****************************************************************************/
		case 170:
		{
/*switch off adjuster vacuum*/
			if( DeloadTimer.Q)
			{
				DeloadStep = 175;
				DeloadTimer.IN = FALSE;
				PlateAtDeloader = PlateAtAdjustedPosition;
				ClearStation(&PlateAtAdjustedPosition);
				break;
			}
			SwitchAdjustTableVacuum(0,ALL,OFF);
			DeloadTimer.IN = TRUE;
			DeloadTimer.PT = AdjusterParameter.TableVacuumOffDelay;
			break;
		}

/* Table to startposition */
		case 175:
		{
			if (DisableTable)
				break;

			if ( FU.cmd_Target == FALSE )
			{
				if( (FU.aktuellePosition_mm < (DeloaderParameter.StartTablePosition)))
					DeloadStep = 182;
				else
				{
					FU.TargetPosition_mm = DeloaderParameter.StartTablePosition;
					FU.cmd_Target = TRUE;
					DeloadStep = 180;
				}
				DeloadTimer.IN = FALSE;
			}
			break;
		}

		case 180:
		{
			if( (abs(FU.aktuellePosition_mm - DeloaderParameter.StartTablePosition) < 1.0)
			 && !FU.cmd_Target
			  )
			{
				DeloadTimer.IN = FALSE;
				DeloadStep = 182;
				break;
			}
			break;
		}
/*liftpins up*/
		case 182:
		{
			if(DeloadTimer.Q)
			{
				DeloadTimer.IN = FALSE;
				DeloadStep = 183;
				break;
			}
			DeloadTimer.IN = !In_LiftingPinsDown;
/* make sure, this code is only executed once */
			if(Out_LiftingPinsDown)
			{
/* pins were down longer than 2 min or first time after power on:
   give them more time
 */
				if(LiftpinsDownTimer.Q || FirstTime)
					DeloadTimer.PT = 500;
				else
					DeloadTimer.PT = 20;
			}
			FirstTime = FALSE;
			Out_LiftingPinsUp = ON;
			Out_LiftingPinsDown = OFF;
			break;
		}

/* Blowair on */
		case 183:
		{
			if (DisableTable)
				break;
/*wait, til conveyor belt free*/
			if( PlateOnConveyorBelt.present)
				break;

			AdjustBlowairOn = ON;
			DeloadTimer.IN = TRUE;
			DeloadTimer.PT = 50;
			DeloadStep = 184;

			break;
		}

/* wait with Blowair on */
		case 184:
		{
			if(DeloadTimer.Q)
			{
				DeloadTimer.IN = FALSE;
				DeloadStep = 185;
			}

			break;
		}

/* Table to endposition */
		case 185:
		{
			if (DisableTable)
				break;
/*wait, til conveyor belt free*/
			if( PlateOnConveyorBelt.present)
				break;

			if ( FU.cmd_Target == FALSE )
			{
				OldParkSpeed = X_Param.ParkSpeed;
				ParkSpeedChanged = TRUE;
				if(ManualMode)
					X_Param.ParkSpeed = DeloaderParameter.TableDeloadSpeedManual;
				else
					X_Param.ParkSpeed = DeloaderParameter.TableDeloadSpeed;
				FU.TargetPosition_mm = DeloaderParameter.EndTablePosition;
				FU.cmd_Target = TRUE;
/*				AdjustBlowairOn = (PlateAtDeloader.PlateConfig != BROADSHEET);*/
				AdjustBlowairOn = ON;
				DeloadTimer.IN = FALSE;
				DeloadStep = 190;
			}
			break;
		}
/* wait for table to arrive in end position, lift pins down on the way, Blowair off when there*/
		case 190:
		{
			if( (FU.aktuellePosition_mm > (DeloaderParameter.StartTablePosition + 50.0) )
			 && !In_LiftingPinsDown)
			{
				Out_LiftingPinsUp = OFF;
				Out_LiftingPinsDown = ON;
			}

			if( (abs(FU.aktuellePosition_mm - DeloaderParameter.EndTablePosition) < 1.0)
			 && !FU.cmd_Target
			  )
			{
				X_Param.ParkSpeed = OldParkSpeed;
				ParkSpeedChanged = FALSE;
				AdjustBlowairOn = OFF;
				DeloadStep = 192;
				break;
			}
			break;
		}
/*liftpins down, should be done in step 190 already, just double check...*/
		case 192:
		{
			if(In_LiftingPinsDown)
			{
				DeloadTimer.IN = FALSE;
				DeloadStep = 200;
				break;
			}
			Out_LiftingPinsUp = OFF;
			Out_LiftingPinsDown = ON;
			break;
		}

		case 200:
		{
			if(MoveToRelPosition(CONVEYORBELT,
			                     350*Motors[CONVEYORBELT].Parameter.IncrementsPerMm,
			                     3000, &ConvMotStep)
			  )
			{
				DeloadTimer.IN = FALSE;
				DeloadStep = 205;
				break;
			}
			break;
		}
		case 205:
		{
			if(Motors[CONVEYORBELT].Moving)
			{
				DeloadTimer.IN = FALSE;
				DeloadStep = 210;
				break;
			}
			break;
		}
		case 210:
		{
			if(!Motors[CONVEYORBELT].Moving)
			{
				DeloadTimer.IN = FALSE;
				AdjustReady = FALSE;
				if(AUTO)
				{
					DeloadReady = TRUE;
					PlateOnConveyorBelt = PlateAtDeloader;
				}
				else
				{
					PlateOnConveyorBelt.present = TRUE;
					PlateOnConveyorBelt.PlateConfig = PlateToDo.PlateConfig;
				}
				ClearStation(&PlateAtDeloader);
				DeloadStep = 0;
				DeloadStart = FALSE;
				break;
			}
			break;
		}
	} /*switch*/

/****************************************************************/
/* CONVEYOR BELT */
/****************************************************************/

/*EGM Fehlermeldung: kein Power-On Signal oder länger keine Einlauffreigabe*/
	EGMErrorDelay.IN = !StatusEGM2 && !GlobalParameter.ProcessorSimulation;
	EGMErrorDelay.PT = DeloaderParameter.EGMStopDelay;
	TON_10ms(&EGMErrorDelay);

	AlarmBitField[22] = (EGMErrorDelay.Q || !StatusEGM1) && !GlobalParameter.ProcessorSimulation;
	AlarmBitField[23] = (!VCP && !GlobalParameter.PunchSimulation);

	if (DeloaderParameter.PinsUpDelay > 999) DeloaderParameter.PinsUpDelay = 999;
	if (DeloaderParameter.PinsDownDelay > 999) DeloaderParameter.PinsDownDelay = 999;

	TON_10ms(&ConveyorBeltTimer);

/*OFF-delay for sensor 200 ms */
	ConveyorBeltSensorDelay1.IN = In_ConveyorBeltSensor[0] || In_ConveyorBeltSensor[1];
	ConveyorBeltSensorDelay1.PT = 20;
	TOF_10ms(&ConveyorBeltSensorDelay1);

/*if flag is reset, stop the sequence*/
	if( !PlateOnConveyorBelt.present )
	{
		ConveyorBeltStep = 0;
	}

	if (!DeloaderParameter.EnableStopPins)
	{
		StopPinsUp = 0;
	}

	switch (ConveyorBeltStep)
	{
		case 0:
		{
			ConveyorBeltTimer.IN = FALSE;
/*Simulation: just delete PlateOnConveyorBelt flag, don't start sequence*/
			if (PlateTransportSim || ConveyorbeltSimulation)
			{
				ClearStation(&PlateOnConveyorBelt);
				break;
			}
/*wait for plate on belt (set by deloading sequence)*/
/*and no plate on sensor*/
			if( !PlateOnConveyorBelt.present) break;

			ConveyorBeltTimer.IN = FALSE;

/*Plate arrived, first thing is: stop pins up (should be the case already...)*/
			if (DeloaderParameter.EnableStopPins)
			{
				StopPinsUp = 1;
			}

			if( (PlateOnConveyorBelt.PlateConfig != PANORAMA)
			 && (PlateOnConveyorBelt.PlateConfig != BROADSHEET) )
			{
				ConveyorBeltTimer.IN = FALSE;
				Out_ConveyorbeltLateral = ON;
				ConveyorBeltStep = 2;
				break;
			}
			else
				ConveyorBeltStep = 5;

			break;
		}

		case 2:
		{
			if(ConveyorBeltTimer.Q)
			{
				Out_ConveyorbeltLateral = OFF;
				ConveyorBeltTimer.IN = FALSE;
				ConveyorBeltStep = 3;
				break;
			}
			ConveyorBeltTimer.IN = TRUE;
			ConveyorBeltTimer.PT = 10;
			Out_ConveyorbeltLateral = ON;
			break;
		}

		case 3:
		{
			if(ConveyorBeltTimer.Q)
			{
				ConveyorBeltTimer.IN = FALSE;
				ConveyorBeltStep = 5;
				break;
			}

			ConveyorBeltTimer.IN = TRUE;
			if( (DeloaderParameter.ConvLateralMoveTime > 0) && (DeloaderParameter.ConvLateralMoveTime < 3000) )
				ConveyorBeltTimer.PT = DeloaderParameter.ConvLateralMoveTime;
			else
				ConveyorBeltTimer.PT = 200;
			break;
		}

		case 5:
		{
/* Start the belt to move plate to the sensor/pins*/

			if( SendMotorCmd(CONVEYORBELT,CMD_MOVE_AT,TRUE,DeloaderParameter.ConveyorBeltSpeed) )
			{
				ConveyorBeltOn = TRUE;
				ConveyorBeltStep = 10;
				ConveyorBeltTimer.IN = TRUE;
				ConveyorBeltTimer.PT = 6000; /*60 sec*/
			}
			break;
		}
		case 10:
		{
/* wait, until plate reaches sensor */
/*measure the time*/
			if (In_ConveyorBeltSensor[0] || In_ConveyorBeltSensor[1])
			{
				if (DeloaderParameter.EnableStopPins)
					ConveyorBeltStep = 15;
				else
				{
/*belt is moving, if processor OK just go on to step 40*/
					if ( ((StatusEGM1 && StatusEGM2) || GlobalParameter.ProcessorSimulation	)
					&&  (VCP || GlobalParameter.PunchSimulation) )
						ConveyorBeltStep = 40;
					else
/*processor not ok -> step 20 to stop belt*/
						ConveyorBeltStep = 20;
				}
				ConveyorBeltTimer.IN = FALSE;
				ConveyorTime = ConveyorBeltTimer.ET;
				break;
			}
/* plate after 60 sec not there -> ERROR */
/*consider it's been taken out*/
			if (ConveyorBeltTimer.Q)
			{
				ConveyorBeltTimer.IN = FALSE;
				ConveyorBeltStep = 55;
			}
			break;
		}
		case 15:
		{
/* wait a little to let plate reach the pins */
			ConveyorBeltTimer.IN = TRUE;
			ConveyorBeltTimer.PT = DeloaderParameter.PinsDownDelay;
			if (ConveyorBeltTimer.Q)
			{
				ConveyorBeltStep = 20;
				ConveyorBeltTimer.IN = FALSE;
			}
			break;
		}

/*Band stoppen*/
		case 20:
		{
			if( SendMotorCmd(CONVEYORBELT,CMD_STOP,FALSE,0L) )
			{
				ConveyorBeltOn = FALSE;
				ConveyorBeltStep = 30;
				ConveyorBeltTimer.IN = FALSE;
			}
			break;
		}

/* 12.07.07 "Slow Mode" */
		case 30:
		{
/* SlowMode aktiviert: Warten*/
			if(SlowMode)
			{
				ConveyorBeltTimer.IN = TRUE;
				ConveyorBeltTimer.PT = GlobalParameter.SlowModeWaitTime;
				ConveyorBeltStep = 31;
			}
			else
			/* kein SlowMode: einfach weiter */
				ConveyorBeltStep = 32;
			break;
		}
/* Warten, bis timer abgelaufen */
		case 31:
		{
			if (ConveyorBeltTimer.Q || !SlowMode)
			{
				ConveyorBeltTimer.IN = FALSE;
				ConveyorBeltStep = 32;
			}
			break;
		}

		case 32:
		{

/*wait for "ready" from Processor*/
/*StatusEGM1 -> Pwr ON*/
/*StatusEGM2 -> Ready*/
			ConveyorBeltTimer.IN = FALSE;
			if ( ((StatusEGM1 && StatusEGM2) || GlobalParameter.ProcessorSimulation	)
			&&  (VCP || GlobalParameter.PunchSimulation) )
				ConveyorBeltStep = 35;
			break;
		}

		case 35:
		{
/* Start the belt to move plate into the processor*/
			if( SendMotorCmd(CONVEYORBELT,CMD_MOVE_AT,TRUE,DeloaderParameter.ConveyorBeltSpeed) )
			{
				ConveyorBeltOn = TRUE;
				ConveyorBeltStep = 36;
				ConveyorBeltTimer.IN = TRUE;
				ConveyorBeltTimer.PT = 4000; /*40 sec*/
			}
			break;
		}

		case 36:
		{
/*wait until plate on sensor (maybe off sensor because it was moved back too far )*/
			if (In_ConveyorBeltSensor[0] || In_ConveyorBeltSensor[1])
			{
				ConveyorBeltTimer.IN = FALSE;
				ConveyorBeltStep = 40;
				break;
			}

/*Error handling: plate doesn't reach sensor in time*/
/*consider it's been taken out*/
			if (ConveyorBeltTimer.Q)
			{
				ConveyorBeltTimer.IN = FALSE;
				ConveyorBeltStep = 55;
			}
			break;
		}

		case 40:
		{
/*wait, until processor signals "not ready" : */
/*now the plate moves into the processor*/

/*StatusEGM1 -> Pwr ON*/
/*StatusEGM2 -> Ready*/
			if ( !StatusEGM2 || GlobalParameter.ProcessorSimulation)
			{
				ConveyorBeltTimer.IN = TRUE;
				ConveyorBeltTimer.PT = 12000; /*120 sec*/
				ConveyorBeltStep = 45;
				InformBluefin();
				break;
			}

/*if sensor becomes free before processor signals "not ready" jump to step 50*/
/*stop waiting for processor*/
			if ( !ConveyorBeltSensorDelay1.Q )
			{
				ConveyorBeltTimer.IN = FALSE;
				ConveyorBeltStep = 50;
				InformBluefin();
				break;
			}

			break;
		}

		case 45:
		{
/*wait until plate off sensor */
			if ( !ConveyorBeltSensorDelay1.Q )
			{
				ConveyorBeltTimer.IN = FALSE;
				ConveyorBeltStep = 50;
				break;
			}

/*Error handling: plate doesn't leave sensor in time*/
			if (ConveyorBeltTimer.Q)
			{
				ConveyorBeltTimer.IN = FALSE;
				ConveyorBeltStep = 55;
			}
			break;
		}

		case 50:
		{
/* no stop pins ->  go on */
			if (!DeloaderParameter.EnableStopPins)
			{
				ConveyorBeltStep = 53;
				ConveyorBeltTimer.IN = FALSE;
				break;
			}

/*wait to let plate be off pins*/
			ConveyorBeltTimer.IN = TRUE;
			ConveyorBeltTimer.PT = DeloaderParameter.PinsUpDelay;
/* after 2 sec: pins up and stop belt*/
			if (ConveyorBeltTimer.Q)
			{
				ConveyorBeltStep = 55;
				if (DeloaderParameter.EnableStopPins)
					StopPinsUp = 1;
			}
			break;
		}

		case 53:
		{
/* wait a little to let plate leave the belt completely */
			ConveyorBeltTimer.IN = TRUE;
/*adjustable time */
			ConveyorBeltTimer.PT = DeloaderParameter.ConveyorBeltDelay;
			if (ConveyorBeltTimer.Q)
			{
				ConveyorBeltStep = 55;
				ConveyorBeltTimer.IN = FALSE;
			}
			break;
		}

/*Band stoppen, Ablauf beendet*/
		case 55:
		{
			if( SendMotorCmd(CONVEYORBELT,CMD_STOP,FALSE,0L) )
			{
				ConveyorBeltOn = FALSE;
				ClearStation(&PlateOnConveyorBelt);
				ConveyorBeltStep = 0;
			}
			break;
		}

	} /* switch (ConveyorBeltStep) */
}
```

- motorfunc.h (reference to Logical/GlobalIncludes/motorfunc.h)

#### motorfunc.c
```c
#ifdef _DEFAULT_INCLUDES
	#include <AsDefault.h>
#endif
/*
                             *******************
******************************* C SOURCE FILE *******************************
**                           *******************                           **
**                                                                         **
** project  : LS JET II                                                    **
** filename : MOTORFUNC.C                                                  **
** version  : 1.02                                                         **
** date     : 07.11.2007                                                   **
**                                                                         **
*****************************************************************************
** Abstract                                                                **
** ========                                                                **
** Implementation of motor control functions (sending commands and         **
** check for positions)                                                    **
**                                                                         **
** Copyright (c) 2007, Krause-Biagosch GmbH                                **
** All rights reserved.                                                    **
**                                                                         **
*****************************************************************************
VERSION HISTORY:
----------------
Version     : 1.00
Date        : 20.10.2006
Revised by  : Herbert Aden
Description : Original version.

Version     : 1.01
Date        : 12.10.2007
Revised by  : Herbert Aden
Description : - a variable for holding the current step in function MoveToAbsPosition
                must now be provided by the caller (a pointer to that var of course!)
              - in Fct. IsPositionOK the check for being in a certain position window
                failed, if that window was 0, i.e. if an exact position is to be found
                the expression "currpos - checkpos < deviation" results in false, so it
                was changed to "currpos - checkpos <= deviation" so that if
                currpos==checkpos the result is still true for deviaition==0

Version     : 1.02
Date        : 07.11.2007
Revised by  : Herbert Aden
Description : - bugfix: in RequestMotorData the var SerialCmd.Request was set TRUE
                unconditionally. Caused sporadic Errormessages for serial comm.

*/
#define _MOTORFUNC_C_SRC

/****************************************************************************/
/**                                                                        **/
/**                           INCLUDE FILES                                **/
/**                                                                        **/
/****************************************************************************/
#include "glob_var.h"
#include "asstring.h"
#include <string.h>

#include "motorfunc.h"

/****************************************************************************/
/**                                                                        **/
/**                       DEFINITIONS AND MACROS                           **/
/**                                                                        **/
/****************************************************************************/
/* NONE */

/****************************************************************************/
/**                                                                        **/
/**                      EXPORTED VARIABLES                                **/
/**                                                                        **/
/****************************************************************************/
/*@checked@*/
_GLOBAL   SerialCmd_Typ       SerialCmd;

/****************************************************************************/
/**                                                                        **/
/**                           GLOBAL VARIABLES                             **/
/**                                                                        **/
/****************************************************************************/
static  BOOL                  Send1Ready = 0;

/****************************************************************************/
/**                                                                        **/
/**                          EXPORTED FUNCTIONS                            **/
/**                                                                        **/
/****************************************************************************/

/****************************************************************************/
/** Send commands to a motor                                                */
/****************************************************************************/
BOOL	SendMotorCmd(const INT pMotor,const char *CmdStr,const BOOL UseValue,const DINT Value)
{
	if(SerialCmd.Send == FALSE) /*wait, till no other sending active*/
	{
		strcpy(SerialCmd.CmdString,CmdStr);
		SerialCmd.UseParameter = UseValue;
		SerialCmd.Parameter = Value;
		if (   (STREQ(CmdStr,CMD_ABSOLUTE_POS))
			|| (STREQ(CmdStr,CMD_RELATIVE_POS))
			|| (STREQ(CmdStr,CMD_MOVE_AT))
		  ) /*bei LA oder LR oder V Refdir verwenden, sonst nicht*/
			SerialCmd.UseRefDirection = TRUE;
		else
			SerialCmd.UseRefDirection = FALSE;

		SerialCmd.SendMotor = pMotor;
		SerialCmd.Send = TRUE;
		return TRUE;
	}
	else
		return FALSE;
}

/****************************************************************************/
/** Request data from a motor                                                */
/****************************************************************************/
BOOL	RequestMotorData(const INT pMotor,const char *CmdString)
{
	if( SerialCmd.Send == TRUE )
		return FALSE;
	else
	{
		SerialCmd.Request = TRUE;
		return SendMotorCmd(pMotor,CmdString,FALSE,0);
	}
}

/****************************************************************************/
/** Check, if a motor is in a certain position window                       */
/****************************************************************************/
BOOL	isPositionOk(const INT Motor,const DINT Pos,const DINT Deviation)
{
	DINT tmp;
	if (labs(Deviation) > 0 )
		tmp = labs(Deviation);
	else	/* if Dev is 0, then use deviation defined in motorparam*/
		tmp = labs(Motors[Motor].Parameter.PositionWindow);

	if( labs( labs(Motors[Motor].Position) - labs(Pos) ) <= tmp )
		return TRUE;
	else
		return FALSE;
}

/****************************************************************************/
/** Check, if a motor is below a certain position                           */
/****************************************************************************/
BOOL	isPositionLowerThan(const INT Motor,DINT Pos)
{
	if( labs(Motors[Motor].Position) < (labs(Pos) ) )
		return TRUE;
	else
		return FALSE;
}

/****************************************************************************/
/** Check, if a motor is above a certain position                           */
/****************************************************************************/
BOOL	isPositionHigherThan(const INT Motor,DINT Pos)
{
	if( labs(Motors[Motor].Position) > (labs(Pos) ) )
		return TRUE;
	else
		return FALSE;
}

/****************************************************************************/
/* send commands to paper remove vertical */
/****************************************************************************/
BOOL	PapRemVerticalCmd(BOOL Config,char *CmdString,BOOL UseValue,DINT Value)
{
	if(Config == LEFT)
		return SendMotorCmd(PAPERREMOVE_VERTICAL, CmdString, UseValue, Value);
	else
	if(Config == RIGHT)
		return SendMotorCmd(PAPERREMOVE_VERTICAL2, CmdString, UseValue, Value);
	else
	if ( Send1Ready == FALSE )
	{
		if( SendMotorCmd(PAPERREMOVE_VERTICAL, CmdString, UseValue, Value) )
			Send1Ready = TRUE;

		return FALSE;
	}
	else
	{
		if( SendMotorCmd(PAPERREMOVE_VERTICAL2, CmdString, UseValue, Value) )
		{
			Send1Ready = FALSE;
			return TRUE;
		}
		return FALSE;
	}
}

/****************************************************************************/
/* Check position of paper remove vertical */
/****************************************************************************/
BOOL	isPapRemVerticalOk(BOOL Config,DINT Pos,UDINT MaxDeviation)
{
	if(Config == LEFT)
		return isPositionOk(PAPERREMOVE_VERTICAL, Pos, MaxDeviation);
	else
	if(Config == RIGHT)
		return isPositionOk(PAPERREMOVE_VERTICAL2, Pos, MaxDeviation);
	else
	if ( isPositionOk(PAPERREMOVE_VERTICAL, Pos, MaxDeviation) )
	{
		if ( isPositionOk(PAPERREMOVE_VERTICAL2, Pos, MaxDeviation) )
			return TRUE;
		else
			return FALSE;
	}
	else
		return FALSE;
}

/****************************************************************************/
/* move motor to an absolute position and wait for motion to start */
/****************************************************************************/
BOOL  MoveToAbsPosition(INT pMotor, DINT Pos, DINT Speed, USINT *pStep)
{
	int step = *pStep;

	BOOL retval = FALSE;

	if (pMotor == 0 && Pos == 0L && Speed == 0L)
	{
		step = 0;
		*pStep = 0;
		return FALSE;
	}

	switch (step)
	{
		case 0:
		{
/* send target position */
			if( SendMotorCmd(pMotor,CMD_ABSOLUTE_POS,TRUE,Pos) )
			{
				if ( Speed == DONT_SEND_SPEED )
					step = 20;
				else
					step = 10;
			}
			retval = FALSE;
			break;
		}
/* set speed */
		case 10:
		{
			if( SendMotorCmd(pMotor,CMD_SPEED,TRUE,Speed) )
			{
				step = 20;
			}
			retval = FALSE;
			break;
		}
		case 20:
		{
/* start motion */
			if( SendMotorCmd(pMotor,CMD_START_MOTION,FALSE,0L) )
			{
				step = 30;
			}
			retval = FALSE;
			break;
		}
		case 30:
		{
/* Wait til motion begins or Motor is in position (might be already there!)*/
			if( Motors[pMotor].Moving
			    ||
			    isPositionOk(pMotor,Pos,0) )
			{
				step = 0;
				retval = TRUE;
			}
			break;
		}
	}
	*pStep = step;
	return retval;
}

/****************************************************************************/
/* move motor to an relative position without waiting for motion to start */
/****************************************************************************/
BOOL  MoveToRelPosition(INT pMotor, DINT Pos, DINT Speed, USINT *pStep)
{
	int step = *pStep;

	BOOL retval = FALSE;

	if (pMotor == 0 && Pos == 0L && Speed == 0L)
	{
		step = 0;
		*pStep = 0;
		return FALSE;
	}

	switch (step)
	{
		case 0:
		{
/* send target position */
			if( SendMotorCmd(pMotor,CMD_RELATIVE_POS,TRUE,Pos) )
			{
				if ( Speed == DONT_SEND_SPEED )
					step = 20;
				else
					step = 10;
			}
			retval = FALSE;
			break;
		}
/* set speed */
		case 10:
		{
			if( SendMotorCmd(pMotor,CMD_SPEED,TRUE,Speed) )
			{
				step = 20;
			}
			retval = FALSE;
			break;
		}
		case 20:
		{
/* start motion */
			if( SendMotorCmd(pMotor,CMD_START_MOTION,FALSE,0L) )
			{
				step = 30;
			}
			retval = FALSE;
			break;
		}
		case 30:
		{
			step = 0;
			retval = TRUE;
			break;
		}
	}
	*pStep = step;
	return retval;
}

/****************************************************************************/
/**                                                                        **/
/**                          LOCAL FUNCTIONS                               **/
/**                                                                        **/
/****************************************************************************/
/* NONE */

/****************************************************************************/
/**                                                                        **/
/**                                 EOF                                    **/
/**                                                                        **/
/****************************************************************************/
```

- glob_var.h (reference to Logical/GlobalIncludes/glob_var.h)

- auxfunc.h (reference to Logical/GlobalIncludes/auxfunc.h)

### Program Logical/Exposer/Ablauf/adjust (ANSIC, version 1.11.0) - Ausrichten

#### ausrichten.c
```c
#ifdef _DEFAULT_INCLUDES
	#include <AsDefault.h>
#endif
/****************************************************************************/
/*	Ablauf Platte Ausrichten */
/*																			*/
/*																			*/
/*	Versionsgeschichte:														*/
/*  Version		Datum		Änderung								von		*/
/*	1.0			16.09.02	erste Implementation					HA		*/
/*	1.1			30.10.02	Wenn Ausrichten fehlschlägt wird nicht 			*/
/*							belichtet								HA		*/
/*	1.11			02.04.03	Fehlermeldung bei Ausrichtfehler	HA		*/
/*																			*/
/*																			*/
/****************************************************************************/

#include "glob_var.h"
#include "asstring.h"
#include "in_out.h"
#include <string.h>
#include "Motorfunc.h"
#include "auxfunc.h"

_LOCAL	USINT	AdjustStep;
_LOCAL TON_10ms_typ AdjustTimer,AddBlowairValveTimer;
USINT			tmp[20];

_GLOBAL	REAL	DropPosition;
_GLOBAL BOOL	AdjustFailed;
_GLOBAL BOOL	StopPlateTaking;
/*HA 07.05.03 V1.06*/
_GLOBAL BOOL	LastPlateIsReady;
/*HA 05.09.03 V1.51 to avoid adjustsensor triggered by deloaded plate*/
_GLOBAL 	BOOL			DisableAdjustSensor;

_LOCAL	USINT	FailCounter;
static USINT MotStep;
static BOOL tmpfail;
static BOOL LeftWasOK,RightWasOK;
static    USINT               PinsStep;       /* holds current step of fct AdjPins */
static    TON_10ms_typ        PinsTimer;

/****************************************************************/
/****************************************************************/
_LOCAL	UINT ManualLoadingStep;
static	TON_10ms_typ ManualLoadingTimer;
_GLOBAL	REAL	TablePosDrop;

/****************************************************************/
/****************************************************************/

_INIT void init(void)
{
	PinsStep = 0;
	PinsTimer.IN = FALSE;
	ManualLoadingStep = 0;
	ManualLoadingStart = FALSE;
	ManualLoadingTimer.IN = FALSE;
	MotStep = 0;
	AdjustStep		= 0;
	AdjustStart	= 0;
	AdjustReady		= 0;
	AdjustTimer.IN	= 0;
	AdjustTimer.PT	= 10; /*just to have any value in there...*/
	AdjustFailed	= 0;
	FailCounter		= 0;
	AddBlowairValveTimer.IN = 0;
	AddBlowairValveTimer.PT = 50;
	return;
}

/****************************************************************************/
/* zyklischer Teil*/
/****************************************************************************/
_CYCLIC void cyclic(void)
{
	SequenceSteps[3] = AdjustStep;

/*validate*/
	if (AdjusterParameter.MaxFailedPlates > 10)
			AdjusterParameter.MaxFailedPlates = 3;
	if ( (AdjusterParameter.AdjustSim != 0)&& (AdjusterParameter.AdjustSim != 1))
		AdjusterParameter.AdjustSim = 0;

	TON_10ms(&AdjustTimer);
	TON_10ms(&ManualLoadingTimer);
	TON_10ms(&PinsTimer);

/* bei Tischblasluft wird jetzt nach 0,5 sec das Vakuumventil zugeschaltet
 * um den Luftdurchsatz zu erhöhen, Option schaltbar durch Parameter
 * "AdjusterParameter.AddBlowairValveDelay" 0->AUS, 1->EIN
*/
	if (AdjusterParameter.AddBlowairValveDelay > 1)
		AdjusterParameter.AddBlowairValveDelay = 1;

	if (AdjusterParameter.AddBlowairValveDelay > 0)
	{
		AddBlowairValveTimer.PT = 50;
		AddBlowairValveTimer.IN = AdjustStart && AdjustBlowairOn;
		TON_10ms(&AddBlowairValveTimer);

		if (AddBlowairValveTimer.Q )
		{
			AdjustVacuumOn[0] = ON;
			AdjustVacuumOn[1] = ON;
		}
	}
/*safety*/
	if( !AdjustStart )
	{
		AdjustStep = 0;
	}

	switch (AdjustStep)
	{
		case 0:
		{
			LeftWasOK = FALSE;
			RightWasOK = FALSE;
			if( !AdjustStart
			 ||  ExposeStart
			 ||  DeloadStart
			 ||  PlateTakingStart
			  )
				break;
/************************************************/
/*
			if( isPositionHigherThan(FEEDER_VERTICAL,
		                            labs(AdjusterParameter.FeederFixposition) + 20L)
			 || PlateTakingStart
		      )
			{
				AdjustStart = FALSE;
		    	break;
		    }
*/
/****************************/

			AdjustTimer.IN = FALSE;
			AdjustReady = FALSE;
			FailCounter = 0;

			if(   In_FeederHorActive
			  && !In_FeederHorInactive
			  &&  Out_FeederHorActive
			  )
				AdjustStep = 200;
			else
				AdjustStep = 2;
			break;
		}

		case 2:
		{
			Out_FeederHorActive = TRUE;
			if(In_FeederHorActive && !In_FeederHorInactive)
				AdjustStep = 200;

			break;
		}

/* Pins up */
		case 200:
		{
			if(AdjPins(PlateAtFeeder.PlateConfig,&PinsStep,&PinsTimer))
				AdjustStep = 202;
			break;
		}

/* Tisch in Übergabepos fahren */
		case 202:
		{
			TablePosDrop = FeederParameter.MinTablePosDrop;

/*Sicherheit: Position prüfen und ggf. begrenzen*/
			if ( TablePosDrop > X_Param.MaxPosition )
			{
				TablePosDrop = X_Param.MaxPosition-1;
			}

/*kann zwar nicht vorkommen, aber sicher ist sicher...*/
			if ( TablePosDrop < X_Param.MinPosition )
				TablePosDrop = X_Param.MinPosition+1;

/*schon da? sollte der Fall sein nach Entladen...*/
			if ( abs(FU.aktuellePosition_mm - TablePosDrop)< 2 )
			{
/*Tisch ist in Position -> OK, weiter*/
				AdjustStep = 5;
				break;
			}
/*noch nicht da, ok, dann hinfahren*/
			if ( FU.cmd_Target == 0 )
			{
				FU.TargetPosition_mm = TablePosDrop;
				FU.cmd_Target = TRUE;
				AdjustStep = 205;
			}
			break;
		}
		case 205:
		{
/*und warten*/
			if( (abs(FU.aktuellePosition_mm - FU.TargetPosition_mm) < 1.0)
			&& 	(FU.cmd_Target == FALSE) )
			{
/*Tisch ist in Position -> OK, weiter*/
				AdjustStep = 5;
			}
			break;
		}

		case 5:
		{
			if(isPositionOk(FEEDER_VERTICAL,AdjusterParameter.FeederAdjustposition,0))
				AdjustStep = 20;
			else
				AdjustStep = 10;
			break;
		}

/* Feeder down onto table */
		case 10:
		{
			if( MoveToAbsPosition(FEEDER_VERTICAL,
			                      AdjusterParameter.FeederAdjustposition,
			                      FeederParameter.SpeedUpFast,
			                      &MotStep) )
			{
				AdjustStep = 20;
				Out_AdjustSignalCross = (PlateAtFeeder.PlateConfig == BROADSHEET);
				AdjustTimer.IN = FALSE;
			}

			break;
		}
/* wait for feeder */
		case 20:
		{
			if(isPositionOk(FEEDER_VERTICAL,AdjusterParameter.FeederAdjustposition,0))
			{
				SwitchFeederVacuum(0,ALL,OFF);
				SwitchAdjustVacuum(PlateAtFeeder.PlateType,PlateAtFeeder.PlateConfig,ON);
				AdjustBlowairOn = ON;
				tmpfail = FALSE;
/* damit die Sauger auch bei Transport Simulation bewegt werden*/
				MoveAdjustSucker(PlateAtFeeder.PlateConfig, ACTIVE);
				AdjustStep = 30;
				LeftWasOK = FALSE;
				RightWasOK = FALSE;
				break;
			}
			break;
		}

		case 30:
		{
			BOOL tmpOK;

			if(PlateAtFeeder.present)
			{
				if(PlateAtFeeder.PlateConfig == BOTH)
				{
					if(AdjustOK(LEFT))
						LeftWasOK = TRUE;
					if(AdjustOK(RIGHT))
						RightWasOK = TRUE;

					tmpOK = LeftWasOK && RightWasOK;
				}
				else
					tmpOK = AdjustOK(PlateAtFeeder.PlateConfig);
			}
			else
				tmpOK = AdjustOK(LEFT);

			if(tmpOK)
			{
				AdjustTimer.IN = FALSE;
				tmpfail = FALSE;
				AdjustStep = 40;
				break;
			}
/* timeout, retry */
			if(AdjustTimer.Q)
			{
				AdjustTimer.IN = FALSE;
				tmpfail = TRUE;
				AdjustStep = 40;
				break;
			}
			MoveAdjustSucker(PlateAtFeeder.PlateConfig, ACTIVE);
			AdjustTimer.IN = TRUE;
			AdjustTimer.PT = AdjusterParameter.TimeoutAdjustedPosition;
			break;
		}

/* Blowair off */
		case 40:
		{
			if(AdjustTimer.Q)
			{
				AdjustTimer.IN = FALSE;
				AdjustStep = 50;
				break;
			}
			AdjustBlowairOn = OFF;
			AdjustTimer.IN = TRUE;
			AdjustTimer.PT = AdjusterParameter.BlowairOffDelay;

			break;
		}
/* Vacuum on */
		case 50:
		{

			if(AdjustTimer.Q)
			{
				AdjustTimer.IN = FALSE;
				AdjustStep = 60;
				break;
			}

			SwitchAdjustTableVacuum(PlateAtFeeder.PlateType,PlateAtFeeder.PlateConfig,ON);
			AdjustTimer.IN = TRUE;
			AdjustTimer.PT = AdjusterParameter.TableVacuumOnDelay;
			break;
		}

		case 60:
		{
/*			if(!CheckAdjustVacuum(0,ALL) || PlateTransportSim)*/
			if(AdjustTimer.Q)
			{
				AdjustTimer.IN = FALSE;
/* adjusting was ok*/
				if(!tmpfail)
				{
					AdjustStep = 130;
					PlateAtAdjustedPosition = PlateAtFeeder;
					break;
				}
				else
					AdjustStep = 70;
				break;
			}
			SwitchAdjustVacuum(0,ALL, OFF);
			AdjustTimer.IN = TRUE;
			AdjustTimer.PT = AdjusterParameter.AdjVacuumOffDelay;

			break;
		}

		case 70:
		{
			if(AdjustTimer.Q)
			{
				AdjustTimer.IN = FALSE;
				FailCounter++;
				if(FailCounter > AdjusterParameter.MaxAttempts)
				{
					SwitchAdjustTableVacuum(0,ALL,OFF);
					AdjustBlowairOn = OFF;
					AdjustStep = 130;
					tmpfail = TRUE;
					StopPlateTaking = 0;
					START = 0;
					FailCounter = 0;

/* HA 15.09.03 V1.60 Adjusting failed: error message */
					AbfrageText1 = 52;
					if(PlateAtFeeder.PlateConfig == BOTH)
					{
						if(!LeftWasOK && !RightWasOK)
							AbfrageText2 = 22;
						else
						if(!LeftWasOK)
							AbfrageText2 = 20;
						else
						if(!RightWasOK)
							AbfrageText2 = 21;
					}
					else
						AbfrageText2 = 0;

					AbfrageText3 = 53;

					if(wBildAktuell != 41 )
						OrgBild = wBildAktuell;
					wBildNeu = 41;
					AbfrageOK = 0;
					AbfrageCancel = 0;
					IgnoreButtons = 1;
					OK_CancelButtonInv = 1;
					OK_ButtonInv = 0;
					AbfrageIcon = CAUTION;
				}
				else
					AdjustStep = 80;

				break;
			}
			MoveAdjustSucker(ALL, INACTIVE);
			AdjustTimer.IN = TRUE;
			AdjustTimer.PT = AdjusterParameter.AdjInactiveTime;
 			break;
		}

/*************************************************************************/
		case 80:
		{
/*			if(CheckAdjustVacuum(PlateAtFeeder.PlateType,PlateAtFeeder.PlateConfig))*/
			if(AdjustTimer.Q)
			{
				AdjustTimer.IN = FALSE;
				AdjustStep = 90;
				break;
			}
			SwitchAdjustVacuum(PlateAtFeeder.PlateType,PlateAtFeeder.PlateConfig,ON);
			AdjustTimer.IN = TRUE;
			AdjustTimer.PT = AdjusterParameter.AdjVacuumOnDelay;
			tmpfail = FALSE;
			break;
		}

		case 90:
		{
			if(AdjustTimer.Q)
			{
				AdjustBlowairOn = ON;
				AdjustTimer.IN = FALSE;
				AdjustStep = 30;
				break;
			}
			SwitchAdjustTableVacuum(0,ALL,OFF);
			AdjustTimer.IN = TRUE;
			AdjustTimer.PT = AdjusterParameter.TableVacuumOffDelay;
			break;
		}
/*************************************************************************/
/* Feeder up */
		case 130:
		{
			if( MoveToAbsPosition(FEEDER_VERTICAL,
			                      FeederParameter.VerticalPositions.Up,
			                      FeederParameter.SpeedUpFast,
			                      &MotStep) )
			{
				AdjustStep = 140;

			}

			break;
		}
/* wait for feeder */
		case 140:
		{
			if(isPositionOk(FEEDER_VERTICAL,FeederParameter.VerticalPositions.Up,0))
			{
				AdjustFailed = tmpfail;
				AlarmBitField[26] = AdjustFailed;
				AdjustReady = !tmpfail;
				ClearStation(&PlateAtFeeder);
				AdjustStep = 150;
				MoveAdjustSucker(ALL, INACTIVE);
				Out_FeederHorActive = FALSE;
				break;
			}
			break;
		}
		case 150:
		{
			if( !Out_FeederHorActive
			 &&  In_FeederHorInactive
			 && !In_FeederHorActive)
			{
				AdjustStart = FALSE;
				AdjustStep = 0;
				break;
			}
			break;
		}

	} /*switch*/
/******************************************************/
/******************************************************/
/* Manual loading */
	switch (ManualLoadingStep)
	{
		case 0:
		{
			if( PaperRemoveStart
			 || PlateTakingStart
			 || AdjustStart
			 || ExposeStart
			 || DeloadStart
			  )
				break;

			if(ManualLoadingStart)
				ManualLoadingStep = 5;
			break;
		}
		case 5:
		{
			if(AdjPins(PlateToDo.PlateConfig,&PinsStep,&PinsTimer))
				ManualLoadingStep = 10;
			break;
		}

		case 10:
		{
/*check, if Feeder is out of collision area (should be the case here)*/
			if( isPositionHigherThan(FEEDER_VERTICAL, labs(AdjusterParameter.FeederAdjustposition) + 50L) )
				break;

			FU.cmd_Park = TRUE;
			ManualLoadingStep = 20;
			break;
		}
		case 20:
		{
			if( (abs(FU.aktuellePosition_mm - X_Param.ParkPosition) < 1.0)
			 && !FU.cmd_Park)
			{
/*				ManualLoadingStep = 30;*/
				ManualLoadingStep = 90;
			}
			break;
		}
		case 30:
		{
			if(!In_ServiceMode)
			{
				ShowMessage(80,81,0,CAUTION,OKONLY,FALSE);
				AbfrageOK = FALSE;
				AbfrageCancel = FALSE;
				ManualLoadingStep = 40;
			}
			else
				ManualLoadingStep = 50;
			break;
		}
		case 40:
		{
			if(AbfrageOK)
			{
				AbfrageOK = FALSE;
				AbfrageCancel = FALSE;
				if(In_ServiceMode)
					ManualLoadingStep = 50;
				else
					ManualLoadingStep = 30;
			}
			break;
		}
		case 50:
		{
			if(In_ServiceMode)
			{
				Out_CoverLockOn = OFF;
				ShowMessage(82,83,84,CAUTION,OKONLY,FALSE);
				AbfrageOK = FALSE;
				ManualLoadingStep = 60;
			}
			break;
		}
		case 60:
		{
			if(AbfrageOK)
			{
				AbfrageOK = FALSE;
				AbfrageCancel = FALSE;
				ManualLoadingStep = 70;
			}
			break;
		}
		case 70:
		{
/* close cover and switch back to auto mode*/
			ShowMessage(85,86,0,CAUTION,OKONLY,FALSE);
			AbfrageOK = FALSE;
			AbfrageCancel = FALSE;
			ManualLoadingStep = 80;
			break;
		}
		case 80:
		{
			if(AbfrageOK)
			{
				AbfrageOK = FALSE;
				AbfrageCancel = FALSE;
				if(!In_ServiceMode)
					ManualLoadingStep = 90;
				else
					ManualLoadingStep = 70;
			}
			break;
		}
		case 90:
		{
			Out_CoverLockOn = ON;
			PlateAtFeeder = PlateToDo;
			ClearStation(&PlateToDo);
			PlateAtFeeder.present = TRUE;
/*			PlateAtFeeder.PlateConfig = BROADSHEET;*/
			PlateAtFeeder.PlateConfig = PANORAMA;
			AdjustStart = TRUE;
			ManualLoadingStep = 0;
			ManualLoadingStart = FALSE;
			break;
		}

	}

	return;
}
```

- motorfunc.h (reference to Logical/GlobalIncludes/motorfunc.h)

- auxfunc.h (reference to Logical/GlobalIncludes/auxfunc.h)

- glob_var.h (reference to Logical/GlobalIncludes/glob_var.h)

### Program Logical/Exposer/Ablauf/aufnahme (ANSIC, version 1.30.0) - Plattenaufnahme
